// ---- _MSG/GVL_MSG_XTS.TcGVL
{attribute 'qualified_only'}
VAR_GLOBAL CONSTANT
  //-----------------------------------------------------------------------------
  // file paths for message system
  //  - compiler define option WIN switches to Windows file paths
  //-----------------------------------------------------------------------------
{IF defined (WIN)}
  {info 'WIN folders'}
  LOG_DIR               : STRING  := 'C:\TwinCAT\#MsgFiles\';       // delimiter at the end is mandatory!!
  CON_DIR               : STRING  := 'C:\TwinCAT\#Configuration\';  // delimiter at the end is mandatory!!
{ELSE}
  {info 'BSD folders'}
  LOG_DIR               : STRING  := '/usr/local/etc/TwinCAT/#MsgFiles/';       // delimiter at the end is mandatory!!
  CON_DIR               : STRING  := '/usr/local/etc/TwinCAT/#Configuration/';  // delimiter at the end is mandatory!!
{END_IF}

  LOG_FILE              : STRING  := 'MSG_XtsTransport_';
  LOG_FILE_APP          : STRING  := 'MSG_Application_';
  LOG_FILE_METRIC       : STRING  := 'MSG_XtsTransportMetrics_';

  MAX_MESSAGE           : UINT    := 2000; // max entry in message list
END_VAR
VAR_GLOBAL
  //-----------------------------------------------------------------------------
  // Message System
  //  - Everybody uses f_MessageSet(ST_Message)
  //    - DECISION WHICH LIST IS MADE IN f_MessageSet !!
  //    - which list to use is determined by e_Device in your message
  //
  //  - MessageData instances are self sufficient and need only 
  //    datafield assignment for correct data-flow
  //
  //
  //-----------------------------------------------------------------------------
  //-----------------------------------------------------------------------------
  //-----------------------------------------------------------------------------
  // (ST_Message.eDevice := e_Device.Application)
  //----------------------------------------------------------------------------- 
  ApplicationMessageData          : fb_MessageDataCtrl;
  ApplicationMessageCtrl          : st_message_ctrl;
  ApplicationMessageState         : st_message_state;

  ApplicationMessages             : ARRAY[1..MAX_MESSAGE] OF ST_Message;
  MessageApplicationIndex         : UINT := 0; // message index for higher layers (grouping, Instances, etc.)
  MessageApplicationError         : UINT := 0; // error counter for higher learning
  //-----------------------------------------------------------------------------
  //-----------------------------------------------------------------------------
  // (ST_Message.eDevice := from Device_Null to XfcAxis)
  //-----------------------------------------------------------------------------
  TransportMessageData            : fb_MessageDataCtrl;
  TransportMessageCtrl            : st_message_ctrl;
  TransportMessageState           : st_message_state;

  TransportMessages               : ARRAY[1..MAX_MESSAGE] OF ST_Message;
  MessageTransportIndex           : UINT := 0; // message index for base layer
  MessageTransportError           : UINT := 0; // error counter for base layer
  //-----------------------------------------------------------------------------
  //-----------------------------------------------------------------------------
  // (ST_Message.eDevice := e_Device.Metrics)
  //-----------------------------------------------------------------------------
  MetricsMessageData              : fb_MessageDataCtrl;
  MetricsMessageCtrl              : st_message_ctrl;
  MetricsMessageState             : st_message_state;

  MetricsMessages                 : ARRAY[1..MAX_MESSAGE] OF ST_Message;
  MessageMetricsIndex             : UINT := 0; // message index for metrics data
  MessageMetricsError             : UINT := 0; // error counter for metrics data
  //-----------------------------------------------------------------------------
  //-----------------------------------------------------------------------------
  // (ST_Message.eDevice := e_Device.ProductData)
  //-----------------------------------------------------------------------------
  ProductMessageData              : fb_MessageDataCtrl;   // This is for you
  ProductMessageCtrl              : st_message_ctrl;
  ProductMessageState             : st_message_state;

  ProductMessages                 : ARRAY[1..MAX_MESSAGE] OF ST_Message;
  MessageProductIndex             : UINT := 0; // message index for your product data
  MessageProductError             : UINT := 0; // error counter for your product data
  //-----------------------------------------------------------------------------
  //-----------------------------------------------------------------------------
  fbLocalTime                     : fb_LocalTime;
  dtLocalTime                     : DT;
  sLocalTime                      : STRING;
  //-----------------------------------------------------------------------------
  //-----------------------------------------------------------------------------
  //-----------------------------------------------------------------------------
  //-----------------------------------------------------------------------------
  MessageLevelXpu                 : E_MessageType;
  MessageLevelStations            : ARRAY[1..MAX_STATION] OF E_MessageType;
  MessageLevelMovers              : ARRAY[1..MAX_MOVER]   OF E_MessageType;

  MessageLevelProcess             : ARRAY[1..MAX_PROCESS] OF E_MessageType;

{IF defined (TEST)}
  {info 'TEST logging enabled'}
  MessageLevel                    : E_MessageType := eMessageinfo; // a lot of messages
{ELSE}
  MessageLevel                    : E_MessageType := eMessageEmpty; // only errors are written into list 
{END_IF}

END_VAR

// ---- _MSG/I_MessageData.TcIO
INTERFACE I_MessageData

PROPERTY DirRoot : POINTER to string(255)
SET
END_SET
END_PROPERTY

PROPERTY ErrorIndex : reference to uint
SET
END_SET
END_PROPERTY

PROPERTY FileRoot : pointer to string(255)
SET
END_SET
END_PROPERTY

PROPERTY LocalTime : pointer to DT
SET
END_SET
END_PROPERTY

PROPERTY MessageIndex : reference to uint
SET
END_SET
END_PROPERTY

PROPERTY MsgList : pointer to ARRAY[1..GVL_MSG_XTS.MAX_MESSAGE] OF st_message
SET
END_SET
END_PROPERTY

END_INTERFACE

// ---- _XML/Configuration/I_Configuration_Station.TcIO
INTERFACE I_Configuration_Station

METHOD Check : BOOL
END_METHOD

METHOD PRIVATE Cmd : E_DATA_STATE
VAR_INPUT
  Ctrl      : E_DATA_CTRL;
END_VAR
END_METHOD

PROPERTY Ctrl : REFERENCE to ST_DATA_CTRL
SET
END_SET
END_PROPERTY

PROPERTY Identity : OTCID
GET
END_GET
SET
END_SET
END_PROPERTY

PROPERTY State : REFERENCE TO ST_DATA_STATE
SET
END_SET
END_PROPERTY

PROPERTY StationParameter : pointer to ARRAY[1..MAX_STATION] OF ST_STATION_PARAMETER
SET
END_SET
END_PROPERTY

END_INTERFACE

// ---- APPLICATION/fb_Simulation.TcPOU
//---------------------------------------------------------------------------------------------------------------
//
//  HAUD 2023.03.27
//
//
//  fb_Simulation
//
//    !!! NOT FOR USE IN PRODUCTION !!! --> build something from your mind, this gets messy if you do not
//
//  - grouping of xts stations to sync start process
//  - nFirst to nLast xts stations are checked for starting process simultaneously
//  - basic preparation of station target index in PrepareTarget()
//  - handshake with station control for mover transport through station
//
//---------------------------------------------------------------------------------------------------------------
// This SOFTWARE is provided as an Exemple by THE PROVIDER "as is" and "with all faults." THE PROVIDER makes no 
// representations or warranties of any kind concerning the safety, suitability, lack of viruses, inaccuracies, 
// typographical errors, or other harmful components of this SOFTWARE. There are inherent dangers in the use of 
// any software, and you are solely responsible for determining whether this SOFTWARE is compatible with your 
// equipment and other software installed on your equipment. You are also solely responsible for the protection 
// of your equipment and backup of your data, and THE PROVIDER will not be liable for any damages you may suffer 
// in connection with using, modifying, or distributing this SOFTWARE.
//---------------------------------------------------------------------------------------------------------------
FUNCTION_BLOCK fb_Simulation
VAR
  _nProcessId                 : UINT;

  _sCheck                     : STRING;
  _tonProcess                 : Tc2_Standard.TON;
  _tProcess                   : TIME := T#500MS;

  _AllStationMoverPerMinute   : UDINT;
  _nMoverCountTotal           : UDINT;

  _tonPartsPerMinute          : Tc2_Standard.TON;

  {attribute 'displaymode':='bin'}
  _wEnter                     : DWORD;
  {attribute 'displaymode':='bin'}
  _wStart                     : DWORD;
  {attribute 'displaymode':='bin'}
  _wOut                       : DWORD;
  {attribute 'displaymode':='bin'}
  _wGone                      : DWORD;
  {attribute 'displaymode':='bin'}
  _wEnableProcess             : DWORD; // bits switch on stations

  {attribute 'displaymode':='bin'}
  _TargetMask                 : BYTE;

  _stCtrl                     : POINTER TO ARRAY[1..MAX_STATION]  OF ST_STATION_CTRL;
  _stState                    : POINTER TO ARRAY[1..MAX_STATION]  OF ST_STATION_STATE;

  // controlling bits from properties used on the outside
  _bNext,
  _bMoverEnter,
  _bMoverOut                  : BOOL;

  // who is included in process
  // _nFirst to _nLast MUST be in closed consecutive order
  _nProcessState,
  _nStation,
  _nStationCount,
  _nFirstStation,
  _nLastStation               : UINT;

  _nTarget,
  _nFirstTarget,
  _nLastTarget                : UINT;

  _nPreparedTarget            : ARRAY[1..MAX_MOVER]  OF UINT;

  _nMoverCountStartOld,
  _nMoverCountEnterOld,
  _nMoverCountEnter,
  _nMoverCountStart,
  _nMoverPerMinute,
  _nMoverCount,
  _nMoverCountOld             : ARRAY[1..MAX_STATION]  OF UDINT;

  _rCheckRangeLow,
  _rCheckRangeHigh            : LREAL; // position range the mover has to be in for infeed or sending to happen.

  _MessageLevel               : E_MessageType;
  _stMsg                      : ST_Message;
END_VAR

METHOD Check : BOOL

IF (_nFirstStation < 1) OR
   (_nFirstStation > MAX_STATION)
THEN
  _sCheck                     := '_nFirstStation out of bounds';
  RETURN;
END_IF

IF (_nLastStation < 1) OR
   (_nLastStation > MAX_STATION)
THEN
  _sCheck                     := '_nLastStation out of bounds';
  RETURN;
END_IF

IF (_nFirstTarget < 1) OR
   (_nFirstTarget > MAX_STATION)
THEN
  _sCheck                     := '_nFirstTarget out of bounds';
  RETURN;
END_IF

IF (_nLastTarget < 1) OR
   (_nLastTarget > MAX_STATION)
THEN
  _sCheck                     := '_nLastTarget out of bounds';
  RETURN;
END_IF

IF NOT (_stCtrl  <> 0)
THEN
  _sCheck                     := '_stCtrl: missing pointer';
  RETURN;
END_IF

IF NOT (_stState <> 0)
THEN
  _sCheck                     := '_stState: missing pointer';
  RETURN;
END_IF


_sCheck                       := TO_STRING(E_PROGRESS.PROGRESS_DONE);
Check                         := TRUE;
END_METHOD

PROPERTY CheckRangeHigh : lreal
GET
CheckRangeHigh := _rCheckRangeHigh;
END_GET
SET
_rCheckRangeHigh := CheckRangeHigh;
END_SET
END_PROPERTY

PROPERTY CheckRangeLow : lreal
GET
CheckRangeLow := _rCheckRangeLow;
END_GET
SET
_rCheckRangeLow := CheckRangeLow;
END_SET
END_PROPERTY

METHOD Cycle
VAR_INST
  _interAllStationsCounter    : UDINT;

  _rtrigProcessEnter,
  _rtrigProcessStart,
  _rtrigProcess       : ARRAY[1..MAX_STATION] OF Tc2_Standard.R_TRIG;

  _k                  : UINT;
  _wEnable            : DWORD;
END_VAR
//-----------------------------------------------------------------------------------------------------------------
IF NOT Check() THEN RETURN; END_IF
//-----------------------------------------------------------------------------------------------------------------
_nStationCount                              := _nLastStation - _nFirstStation + 1;
//-----------------------------------------------------------------------------------------------------------------
//-----------------------------------------------------------------------------------------------------------------
IF (_nStationCount < 1)
THEN
  RETURN;
END_IF
//-----------------------------------------------------------------------------------------------------------------
//-----------------------------------------------------------------------------------------------------------------
FOR _nStation := _nLastStation TO _nFirstStation BY(-1) 
DO
  CASE _stState^[_nStation].State
  OF
    //-------------------------------------------------------------------------------------------------------------
    E_STATION_STATE.STATION_DISABLE,
    E_STATION_STATE.STATION_ENABLE, 
    E_STATION_STATE.STATION_DETECT_MOVER:
      _wStart   := _wOut    := _wGone       := 0;
      _wEnter                               := DelBit(_wEnter, (_nStation-_nFirstStation));
      IF (GetBit(_wEnableProcess, (_nStation-_nFirstStation)))
      THEN
        IF (_bMoverEnter)
        THEN
          _stCtrl^[_nStation].Cmd           := E_STATION_CTRL.STATION_ENABLE;
        ELSE
          _stCtrl^[_nStation].Cmd           := E_STATION_CTRL.STATION_DISABLE;
        END_IF
      ELSE
        _stCtrl^[_nStation].Cmd             := E_STATION_CTRL.STATION_DISABLE;
      END_IF


    //-------------------------------------------------------------------------------------------------------------
    E_STATION_STATE.STATION_MOVER_ENTER:
      _wEnter                               := SetBit(_wEnter, (_nStation-_nFirstStation));
      IF _bMoverEnter
      THEN
        _tonProcess(IN                      := FALSE, 
                    PT                      := _tProcess);

        _stCtrl^[_nStation].nTargetStation  := 0;

        IF (_tProcess < T#10MS)
        THEN
          IF (_rCheckRangeHigh > _rCheckRangeLow)
          THEN
            IF (_stState^[_nStation].rMoverModPos > _rCheckRangeLow) AND
               (_stState^[_nStation].rMoverModPos < _rCheckRangeHigh)
            THEN
              _stCtrl^[_nStation].Cmd       := E_STATION_CTRL.STATION_MOVER_SEND;
            END_IF
          ELSE
            IF (_stState^[_nStation].rMoverModPos > _rCheckRangeLow) OR
               (_stState^[_nStation].rMoverModPos < _rCheckRangeHigh)
            THEN
              _stCtrl^[_nStation].Cmd       := E_STATION_CTRL.STATION_MOVER_SEND;
            END_IF
          END_IF
        ELSE
          IF (_rCheckRangeHigh > _rCheckRangeLow)
          THEN
            IF (_stState^[_nStation].rMoverModPos > _rCheckRangeLow) AND
               (_stState^[_nStation].rMoverModPos < _rCheckRangeHigh)
            THEN
              _stCtrl^[_nStation].Cmd       := E_STATION_CTRL.STATION_MOVER_ENTER;
            END_IF
          ELSE
            IF (_stState^[_nStation].rMoverModPos > _rCheckRangeLow) OR
               (_stState^[_nStation].rMoverModPos < _rCheckRangeHigh)
            THEN
              _stCtrl^[_nStation].Cmd       := E_STATION_CTRL.STATION_MOVER_ENTER;
            END_IF
          END_IF
        END_IF
      END_IF

    //-------------------------------------------------------------------------------------------------------------
    E_STATION_STATE.STATION_PROCESS_START:
      _wEnter                               := DelBit(_wEnter, (_nStation-_nFirstStation));
      _wStart                               := SetBit(_wStart, (_nStation-_nFirstStation));
  
      // check if ALL XtsStations have mover in place to work
      IF (_wStart = _wEnableProcess)
      THEN
        _tonProcess(IN                      := TRUE, 
                    PT                      := _tProcess);

        IF _tonProcess.Q
        THEN
          PrepareTargets(FALSE);
          _stCtrl^[_nStation].Cmd           := E_STATION_CTRL.STATION_PROCESS_DONE;
        END_IF
      END_IF

    //-------------------------------------------------------------------------------------------------------------
    E_STATION_STATE.STATION_CHECK_NEST:
      _wEnter                               := SetBit(_wEnter, (_nStation-_nFirstStation));
      _wStart                               := DelBit(_wStart, (_nStation-_nFirstStation));
      _tonProcess(IN                        := FALSE, 
                  PT                        := _tProcess);

      IF (_bNext)
      THEN
        // check if ALL XtsStations have nest to work
        IF (_wEnter = _wEnableProcess)
        THEN
          _stCtrl^[_nStation].Cmd           := E_STATION_CTRL.STATION_MOVER_ENTER;
        END_IF
      END_IF

    //-------------------------------------------------------------------------------------------------------------
    E_STATION_STATE.STATION_MOVER_OUT:
      _wOut                                 := SetBit(_wOut, (_nStation-_nFirstStation));
      _tonProcess(IN                        := FALSE, 
                  PT                        := _tProcess);

      IF _bMoverOut
      THEN
        // nest mask for this mover in target station, sender decides what to work in target
        _stCtrl^[_nStation].nMask           := _TargetMask;

        // check if ALL XtsStations have mover to send
        IF (_wOut = _wEnableProcess)
        THEN
          _nProcessState                    := 10;
        END_IF
      END_IF
  END_CASE
END_FOR
//-----------------------------------------------------------------------------------------------------------------
//-----------------------------------------------------------------------------------------------------------------
CASE _nProcessState
OF
10:
  // ctrl has to decide where to send mover; this depends on YOUR decision
  IF PrepareTargets(TRUE)
  THEN
    PrepareTargets(FALSE);
    _nProcessState                          := 30;
  END_IF
END_CASE
CASE _nProcessState
OF
30:
  FOR _nStation := _nLastStation TO _nFirstStation BY(-1) 
  DO
    IF _bNext
    THEN
      // start outfeed of mover
      _stCtrl^[_nStation].Cmd               := E_STATION_CTRL.STATION_MOVER_OUT;
    END_IF

    CASE _stState^[_nStation].State
    OF
      E_STATION_STATE.STATION_MOVER_GONE:
        _wStart   := _wEnter                := 0;
        // whO is gone?
        _wGone                              := SetBit(_wGone, (_nStation-_nFirstStation));
    END_CASE
  END_FOR
  // check if ALL XtsStations are empty
  IF (_wGone = _wEnableProcess)
  THEN
    _nProcessState                          := 40;
    IF (_MessageLevel > E_MessageType.eMessageVerbose)
    THEN
      _stMsg.eType                          := E_MessageType.eMessageSentient;
      _stMsg.eDevice                        := e_Device.Metrics + TO_UINT(_nProcessId);
      _stMsg.eSubdevice                     := e_Subdevice.Process_StationCollector;
      _stMsg.iErrorNumber                   := _nProcessId;
      _stMsg.sText                          := concat('ALL MOVER: ', TO_STRING(E_STATION_STATE.STATION_MOVER_GONE));

      f_MessageSet(_stMsg);
    END_IF
  END_IF
END_CASE
CASE _nProcessState
OF
40:
  _nProcessState                            := 0;
  FOR _nStation := _nLastStation TO _nFirstStation BY(-1) 
  DO
    // let XtsStations jump back to disable
    _stCtrl^[_nStation].Cmd                 := E_STATION_CTRL.STATION_MOVER_GONE;
  END_FOR
END_CASE
//-----------------------------------------------------------------------------------------------------------------
//-----------------------------------------------------------------------------------------------------------------
//-----------------------------------------------------------------------------------------------------------------
// Mover per Minute counter all XtsStations in range
//-----------------------------------------------------------------------------------------------------------------
_nMoverCountTotal                           :=
_AllStationMoverPerMinute                   := 0; 
//-----------------------------------------------------------------------------------------------------------------
// mover counter
//-----------------------------------------------------------------------------------------------------------------
FOR _k := _nLastStation TO _nFirstStation BY(-1)
DO
  //---------------------------------------------------------------------------------------------------------------
  _rtrigProcess[_k](CLK:= ( _stCtrl^[_k].Cmd = E_STATION_CTRL.STATION_MOVER_OUT));
  //---------------------------------------------------------------------------------------------------------------
  IF _rtrigProcess[_k].Q
  THEN
    _nMoverCount[_k]                        := _nMoverCount[_k] + 1;

    IF (_MessageLevel > E_MessageType.eMessageError)
    THEN
      _stMsg.eType                          := E_MessageType.eMessageInfo;
      _stMsg.eDevice                        := e_Device.Metrics + TO_UINT(_nProcessId);
      _stMsg.eSubdevice                     := e_Subdevice.Process_StationCollector;
      _stMsg.iErrorNumber                   := _k;
      _stMsg.sText                          := concat('MoverCountStation[ ]: ', TO_STRING(_nMoverCount[_k]));
      _stMsg.sText                          := concat(_stMsg.sText, ': E_STATION_CTRL.');
      _stMsg.sText                          := concat(_stMsg.sText, TO_STRING(_stCtrl^[_k].Cmd));
      f_MessageSet(_stMsg);
    END_IF
  END_IF

  //---------------------------------------------------------------------------------------------------------------
  _rtrigProcessStart[_k](CLK:= ( _stState^[_k].State = E_STATION_STATE.STATION_PROCESS_START));
  //---------------------------------------------------------------------------------------------------------------
  IF _rtrigProcessStart[_k].Q
  THEN
    _nMoverCountStart[_k]                   := _nMoverCountStart[_k] + 1;

    IF (_MessageLevel > E_MessageType.eMessageInfo)
    THEN
      _stMsg.eType                          := E_MessageType.eMessageVerbose;
      _stMsg.eDevice                        := e_Device.Metrics + TO_UINT(_nProcessId);
                            
      _stMsg.eSubdevice                     := e_Subdevice.Process_StationCollector;
      _stMsg.iErrorNumber                   := _k;
      _stMsg.sText                          := concat('MoverCountStation[ ]: ', TO_STRING(_nMoverCountEnter[_k]));
      _stMsg.sText                          := concat(_stMsg.sText, ': E_STATION_STATE.');
      _stMsg.sText                          := concat(_stMsg.sText, TO_STRING(_stState^[_k].State));
      f_MessageSet(_stMsg);
    END_IF
  END_IF

  //---------------------------------------------------------------------------------------------------------------
  _rtrigProcessEnter[_k](CLK:= ( _stCtrl^[_k].Cmd = E_STATION_CTRL.STATION_MOVER_ENTER));
  //---------------------------------------------------------------------------------------------------------------
  IF _rtrigProcessEnter[_k].Q
  THEN
    _nMoverCountEnter[_k]                   := _nMoverCountEnter[_k] + 1;

    IF (_MessageLevel > E_MessageType.eMessageVerbose)
    THEN
      _stMsg.eType                          := E_MessageType.eMessageSentient;
      _stMsg.eDevice                        := e_Device.Metrics + TO_UINT(_nProcessId);
                            
      _stMsg.eSubdevice                     := e_Subdevice.Process_StationCollector;
      _stMsg.iErrorNumber                   := _k;
      _stMsg.sText                          := concat('MoverCountStation[ ]: ', TO_STRING(_nMoverCountEnter[_k]));
      _stMsg.sText                          := concat(_stMsg.sText, ': E_STATION_CTRL.');
      _stMsg.sText                          := concat(_stMsg.sText, TO_STRING(_stCtrl^[_k].Cmd));
      f_MessageSet(_stMsg);
    END_IF
  END_IF
  //---------------------------------------------------------------------------------------------------------------
  //---------------------------------------------------------------------------------------------------------------
  IF _tonPartsperMinute.Q
  THEN
    // count every XtsStation in range
    _nMoverPerMinute[_k]                    := _nMoverCount[_k] - _nMoverCountOld[_k];
    _nMoverCountOld [_k]                    := _nMoverCount[_k];

    _nMoverCountEnterOld [_k]               := _nMoverCountEnter[_k];
    _nMoverCountStartOld [_k]               := _nMoverCountStart[_k];
  END_IF
  // sum up all XtsStations in range
  _AllStationMoverPerMinute                 := _AllStationMoverPerMinute + _nMoverPerMinute[_k]; 
  _interAllStationsCounter                  := _AllStationMoverPerMinute + _nMoverPerMinute[_k];

  // sum up all mover counts in range
  _nMoverCountTotal                         := _nMoverCountTotal + _nMoverCount[_k];
END_FOR
//-----------------------------------------------------------------------------------------------------------------
//-----------------------------------------------------------------------------------------------------------------
// total mover per minute message for all stations in this process
//-----------------------------------------------------------------------------------------------------------------
//-----------------------------------------------------------------------------------------------------------------
IF _tonPartsperMinute.q
THEN
  _tonPartsperMinute(IN:=FALSE);

  IF (_MessageLevel > E_MessageType.eMessageError)
  THEN
    _stMsg.eType                          := E_MessageType.eMessageBatch;
    _stMsg.eDevice                        := e_Device.Metrics + TO_UINT(_nProcessId);
  
    _stMsg.eSubdevice                     := e_Subdevice.Process_StationCollector;
    _stMsg.iErrorNumber                   := _nMoverCountTotal;
    _stMsg.sText                          := concat('MoverCountTotal: ', TO_STRING(_nMoverCountTotal));
    _stMsg.sText                          := concat(_stMsg.sText, ': StationLast: ');
    _stMsg.sText                          := concat(_stMsg.sText, TO_STRING(_nLastStation));
    _stMsg.sText                          := concat(_stMsg.sText, ': StationFirst: ');
    _stMsg.sText                          := concat(_stMsg.sText, TO_STRING(_nFirstStation));
    f_MessageSet(_stMsg);
  END_IF
END_IF
//-----------------------------------------------------------------------------------------------------------------
_tonPartsperMinute(IN:= TRUE,   PT:= T#60S);
//-----------------------------------------------------------------------------------------------------------------
//-----------------------------------------------------------------------------------------------------------------
END_METHOD

METHOD PUBLIC DelBit : DWORD
VAR_INPUT
  inVal   : DWORD;
  bitNo   : DINT;
END_VAR
VAR
  wConst : dWORD := 1;
END_VAR
IF ( inVal AND SHL( wConst,bitNo MOD 32 ) ) > 0 THEN
  DelBit := inVal XOR (SHL( wConst,bitNo MOD 32 ));
ELSE
  DelBit := inVal;
END_IF
END_METHOD

METHOD Disable : BOOL
VAR_INPUT
END_VAR
IF NOT (_nLastStation   > 0) OR
   NOT (_nFirstStation  > 0) OR
   NOT (_nLastStation   < MAX_STATION+1) OR
   NOT (_nFirstStation  < MAX_STATION+1)
THEN
  Disable := FALSE;
ELSE
  FOR _nStation := _nLastStation TO _nFirstStation BY(-1) 
  DO
    _stCtrl^[_nStation].Cmd               := E_STATION_CTRL.STATION_DISABLE;
    _stCtrl^[_nStation].nMask             := 0;
  END_FOR

  memset(ADR(_nMoverCount),    0, SIZEOF(_nMoverCount));
  memset(ADR(_nMoverCountOld), 0, SIZEOF(_nMoverCountOld));
  _nProcessState :=  _nTarget             := 0;
  
  Disable := TRUE;
END_IF
END_METHOD

PROPERTY EnableProcess : dword
GET
EnableProcess := _wEnableProcess;
END_GET
SET
_wEnableProcess := EnableProcess;
END_SET
END_PROPERTY

METHOD PUBLIC GetBit : BOOL
VAR_INPUT
  inVal   : DWORD;
  bitNo   : DINT;
END_VAR
VAR
  wConst : DWORD := 1;
END_VAR
IF ( inVal AND SHL( wConst,DINT_TO_SINT(bitNo) MOD 32 ) ) > 0
THEN
  GetBit := TRUE;
ELSE
  GetBit := FALSE;
END_IF
END_METHOD

METHOD Init : BOOL
VAR_INPUT
END_VAR
IF NOT (_nLastStation   > 0) OR
   NOT (_nFirstStation  > 0) OR
   NOT (_nLastStation   < MAX_STATION+1) OR
   NOT (_nFirstStation  < MAX_STATION+1)
THEN
  Init := FALSE;
ELSE
  FOR _nStation := _nLastStation TO _nFirstStation BY(-1) 
  DO
    _stCtrl^[_nStation].Cmd               := E_STATION_CTRL.STATION_INIT;
    _stCtrl^[_nStation].nMask             := 0;
  END_FOR

  memset(ADR(_nMoverCount),    0, SIZEOF(_nMoverCount));
  memset(ADR(_nMoverCountOld), 0, SIZEOF(_nMoverCountOld));
  _nProcessState :=  _nTarget             := 0;
  
  Init := TRUE;
END_IF
END_METHOD

PROPERTY MessageLevel : e_MessageType
GET
MessageLevel := _MessageLevel;
END_GET
SET
VAR
  _ix : uint;
END_VAR
_MessageLevel := MessageLevel;
END_SET
END_PROPERTY

PROPERTY MoverEnter : bool
GET
MoverEnter := _bMoverEnter;
END_GET
SET
_bMoverEnter := MoverEnter;
END_SET
END_PROPERTY

PROPERTY MoverOut : bool
GET
MoverOut := _bMoverOut;
END_GET
SET
_bMoverOut := MoverOut;
END_SET
END_PROPERTY

METHOD Next : BOOL
VAR_INPUT
  Nxt  : Bool;
END_VAR
_bNext := Nxt;
END_METHOD

METHOD PRIVATE PrepareTargets : BOOL
VAR_INPUT
  Execute         : BOOL;
END_VAR
VAR_INST
  _idxStations    : uint;
  _nt,
  _nstate         : UINT;
END_VAR

IF NOT Check() THEN RETURN; END_IF

IF NOT Execute
THEN
  _nstate                             := 0;
END_IF


CASE _nstate
OF
  0:
    IF Execute
    THEN
      _nstate                         := 10;
    END_IF
END_CASE
CASE _nstate
OF
  10:
    _nstate                           := 20;

    FOR _idxStations := _nLastStation TO _nFirstStation BY(-1) 
    DO
      _nt                               := TO_USINT(_nLastTarget - _nTarget);
      _nTarget                          := _nTarget + 1;
  
      _nPreparedTarget[_stState^[_idxStations].nMoverId]  := _nt;
      _stCtrl^[_idxStations].nTargetStation               := TO_USINT(_nt);
  
      IF (_nLastTarget - _nTarget < _nFirstTarget)
      THEN
        _nTarget                        := 0;
      END_IF
    END_FOR
END_CASE
CASE _nstate
OF
  20:
    PrepareTargets                    := TRUE;
END_CASE
END_METHOD

PROPERTY ProcessId : uint
GET
ProcessId := _nProcessId;
END_GET
SET
_nProcessId := ProcessId;
END_SET
END_PROPERTY

PROPERTY ProcessTime : time
GET
ProcessTime := _tProcess;
END_GET
SET
_tProcess := ProcessTime;
END_SET
END_PROPERTY

METHOD PUBLIC SetBit : DWORD
VAR_INPUT
  inVal   : DWORD;
  bitNo   : DINT;
END_VAR
VAR
  wConst  : dWORD := 1;
END_VAR
SetBit := inVal OR SHL( wConst,bitNo MOD 32 );
END_METHOD

PROPERTY StationCount : uint
GET
StationCount := _nStationCount;
END_GET
END_PROPERTY

PROPERTY StationCtrl : pointer to ARRAY[1..MAX_STATION]  OF ST_STATION_CTRL;
SET
_stCtrl := StationCtrl;
END_SET
END_PROPERTY

PROPERTY StationFirst : uint
GET
StationFirst := _nFirstStation;
END_GET
SET
_nFirstStation := StationFirst;
END_SET
END_PROPERTY

PROPERTY StationLast : uint
GET
StationLast := _nLastStation;
END_GET
SET
_nLastStation := StationLast;
END_SET
END_PROPERTY

PROPERTY StationState : POINTER TO ARRAY[1..MAX_STATION]  OF ST_STATION_STATE
SET
_stState := StationState;
END_SET
END_PROPERTY

PROPERTY TargetFirst : uint
GET
TargetFirst := _nFirstTarget;
END_GET
SET
_nFirstTarget := TargetFirst;
END_SET
END_PROPERTY

PROPERTY TargetLast : uint
GET
TargetLast := _nLastTarget;
END_GET
SET
_nLastTarget := TargetLast;
END_SET
END_PROPERTY

PROPERTY TargetMask : byte
GET
TargetMask := _TargetMask;
END_GET
SET
_TargetMask := TargetMask;
END_SET
END_PROPERTY

END_FUNCTION_BLOCK

// ---- _MSG/f_MessageSet.TcPOU
FUNCTION f_MessageSet : BOOL
VAR_INPUT
  stMessage     : ST_Message;
END_VAR
VAR
  _uiIndex      : UINT;
  _MainDevice   : e_Device;
  _nModRes      : UDINT;     // residual after modulo
END_VAR

stMessage.tTime                     := GVL_MSG_XTS.sLocalTime;

// why here? so all calls to this function may stay the same
_nModRes                            := stMessage.eDevice MOD e_Device.General;
_MainDevice                         := stMessage.eDevice - _nModRes;

CASE _MainDevice
OF
  //--------------------------------------------------------------------------------
  e_device.DataProduct:
    // this is your data, if you choose to use this message system
    FOR _uiIndex := 1 TO GVL_MSG_XTS.MAX_MESSAGE
    DO
      IF (GVL_MSG_XTS.ProductMessages[_uiIndex].eType = e_MessageType.eMessageEmpty)
      THEN
        GVL_MSG_XTS.ProductMessages[_uiIndex]      := stMessage;
        GVL_MSG_XTS.MessageProductIndex            := _uiIndex;
        EXIT;
      END_IF
    END_FOR
  
    IF (stMessage.eType = E_MessageType.eMessageError)
    THEN
      // in case of error: increment counter
      GVL_MSG_XTS.MessageProductError              := GVL_MSG_XTS.MessageProductError + 1;
    END_IF
  //--------------------------------------------------------------------------------
  e_Device.Process,
  e_Device.Application:
    FOR _uiIndex := 1 TO GVL_MSG_XTS.MAX_MESSAGE
    DO
      IF (GVL_MSG_XTS.ApplicationMessages[_uiIndex].eType = e_MessageType.eMessageEmpty)
      THEN
        GVL_MSG_XTS.ApplicationMessages[_uiIndex]  := stMessage;    // yes, we grab global values directly, only here
        GVL_MSG_XTS.MessageApplicationIndex        := _uiIndex;
        EXIT;
      END_IF
    END_FOR
    IF (stMessage.eType = E_MessageType.eMessageError)
    THEN
      // in case of error: increment counter
      GVL_MSG_XTS.MessageApplicationError          := GVL_MSG_XTS.MessageApplicationError + 1;
    END_IF
  //--------------------------------------------------------------------------------
  e_Device.MetricsXts:
    FOR _uiIndex := 1 TO GVL_MSG_XTS.MAX_MESSAGE
    DO
      IF (GVL_MSG_XTS.MetricsMessages[_uiIndex].eType = e_MessageType.eMessageEmpty)
      THEN
        GVL_MSG_XTS.MetricsMessages[_uiIndex]      := stMessage;    // yes, we grab global values directly, only here
        GVL_MSG_XTS.MessageMetricsIndex            := _uiIndex;
        EXIT;
      END_IF
    END_FOR
    IF (stMessage.eType = E_MessageType.eMessageError)
    THEN
      // in case of error: increment counter
      GVL_MSG_XTS.MessageMetricsError              := GVL_MSG_XTS.MessageMetricsError + 1;
    END_IF
  //--------------------------------------------------------------------------------
  e_Device.MetricsAxis:
    FOR _uiIndex := 1 TO GVL_MSG_XTS.MAX_MESSAGE
    DO
      IF (GVL_MSG_AXIS.MetricMessages[_uiIndex].eType = e_MessageType.eMessageEmpty)
      THEN
        GVL_MSG_AXIS.MetricMessages[_uiIndex]  := stMessage;    // yes, we grab global values directly, only here
        GVL_MSG_AXIS.MessageMetricIndex        := _uiIndex;
        EXIT;
      END_IF
    END_FOR
    IF (stMessage.eType = E_MessageType.eMessageError)
    THEN
      // in case of error: increment counter
      GVL_MSG_AXIS.MessageMetricError          := GVL_MSG_AXIS.MessageMetricError + 1;
    END_IF
  //--------------------------------------------------------------------------------
  e_Device.Axis,
  e_Device.XfcAxis,
  e_device.XfcTouchProbe,
  e_device.XfcTriggerBox,
  e_Device.Camming,
  e_device.NciChannel,
  e_device.NciChannelCtrl:
    FOR _uiIndex := 1 TO GVL_MSG_XTS.MAX_MESSAGE
    DO
      IF (GVL_MSG_AXIS.MotionMessages[_uiIndex].eType = e_MessageType.eMessageEmpty)
      THEN
        GVL_MSG_AXIS.MotionMessages[_uiIndex]  := stMessage;    // yes, we grab global values directly, only here
        GVL_MSG_AXIS.MessageMotionIndex        := _uiIndex;
        EXIT;
      END_IF
    END_FOR
    IF (stMessage.eType = E_MessageType.eMessageError)
    THEN
      // in case of error: increment counter
      GVL_MSG_AXIS.MessageMotionError           := GVL_MSG_AXIS.MessageMotionError + 1;
    END_IF
  //--------------------------------------------------------------------------------
ELSE
  CASE stMessage.eDevice
  OF
    Device_MainApplication,
    Device_XmlData,              
    Device_Utilities:
      FOR _uiIndex := 1 TO GVL_MSG_XTS.MAX_MESSAGE
      DO
        IF (GVL_MSG_XTS.ApplicationMessages[_uiIndex].eType = e_MessageType.eMessageEmpty)
        THEN
          GVL_MSG_XTS.ApplicationMessages[_uiIndex]:= stMessage;    // yes, we grab global values directly, only here
          GVL_MSG_XTS.MessageApplicationIndex      := _uiIndex;
          EXIT;
        END_IF
      END_FOR
      IF (stMessage.eType = E_MessageType.eMessageError)
      THEN
        // in case of error: increment counter
        GVL_MSG_XTS.MessageApplicationError        := GVL_MSG_XTS.MessageApplicationError + 1;
      END_IF

    Device_MainAxis,
    Device_Nci,
    Device_Cam,
    Device_Functions,
    Device_FlyingSaw,
    Device_ParameterSelector:     // PLC_MOTION
      FOR _uiIndex := 1 TO GVL_MSG_XTS.MAX_MESSAGE
      DO
        IF (GVL_MSG_AXIS.MotionMessages[_uiIndex].eType = e_MessageType.eMessageEmpty)
        THEN
          GVL_MSG_AXIS.MotionMessages[_uiIndex]:= stMessage;    // yes, we grab global values directly, only here
          GVL_MSG_AXIS.MessageMotionIndex      := _uiIndex;
          EXIT;
        END_IF
      END_FOR
      IF (stMessage.eType = E_MessageType.eMessageError)
      THEN
        // in case of error: increment counter
        GVL_MSG_AXIS.MessageMotionError        := GVL_MSG_AXIS.MessageMotionError + 1;
      END_IF

    Device_Main,
    Device_MoverSelector:
      FOR _uiIndex := 1 TO GVL_MSG_XTS.MAX_MESSAGE
      DO
        IF (GVL_MSG_XTS.TransportMessages[_uiIndex].eType = e_MessageType.eMessageEmpty)
        THEN
          GVL_MSG_XTS.TransportMessages[_uiIndex]  := stMessage;
          GVL_MSG_XTS.MessageTransportIndex        := _uiIndex;
          EXIT;
        END_IF
      END_FOR
  ELSE    
    //--------------------------------------------------------------------------------
    FOR _uiIndex := 1 TO GVL_MSG_XTS.MAX_MESSAGE
    DO
      IF (GVL_MSG_XTS.TransportMessages[_uiIndex].eType = e_MessageType.eMessageEmpty)
      THEN
        GVL_MSG_XTS.TransportMessages[_uiIndex]    := stMessage;
        GVL_MSG_XTS.MessageTransportIndex          := _uiIndex;
        EXIT;
      END_IF
    END_FOR
  
    IF (stMessage.eType = E_MessageType.eMessageError)
    THEN
      // in case of error: increment counter
      GVL_MSG_XTS.MessageTransportError := GVL_MSG_XTS.MessageTransportError + 1;
    END_IF
  END_CASE
END_CASE

END_FUNCTION

// ---- _MSG/class/fb_MessageDataCtrl.TcPOU
FUNCTION_BLOCK fb_MessageDataCtrl EXTENDS fb_MessageData
VAR
  _stCtrl       : REFERENCE TO ST_MESSAGE_CTRL;
  _stState      : REFERENCE TO ST_MESSAGE_STATE;

  _eCmd,
  _eCmdOld      : E_MESSAGE_CTRL;

  _eResult,
  _eJobResult   : E_PROGRESS;

  _eState       : E_MESSAGE_STATE;

END_VAR

//-----------------------------------------------------------------------------
// check pointers
//-----------------------------------------------------------------------------
IF NOT Check()
THEN
  _eResult                      := E_PROGRESS.PROGRESS_ERROR;
  RETURN;
END_IF
//-----------------------------------------------------------------------------
// check date
// new message file for a new day
//-----------------------------------------------------------------------------
IF (FolderDate(_dtLocalTime) <> _sFolderDate)
THEN
  _bFileCreated                 := FALSE;
END_IF
//-----------------------------------------------------------------------------
//----------------------------------------------------------------------------- 
// copy to local for debug
_eCmd                         := _stCtrl.Cmd;

// cyclic check for command change
// get state for cmd
IF (_eCmd <> _eCmdOld)
THEN
  // get matching sdtate for Ctrl.Cmd
  _eState                     := Cmd(_eCmd);
  _eCmdOld                    := _eCmd;
END_IF


CASE _eResult
OF
  E_PROGRESS.PROGRESS_INVALID:
    _stState.State            := E_MESSAGE_STATE.MSG_STATE_NULL;

  E_PROGRESS.PROGRESS_ERROR:
    _stState.State            := _eState + E_PROGRESS.PROGRESS_ERROR;

  E_PROGRESS.PROGRESS_DONE:
    _stState.State            := _eState + E_PROGRESS.PROGRESS_DONE;

ELSE
  // work in progress
  // update progress for extern use
  _stState.State              := _eState + _eResult;

  CASE _eState
  OF
    E_MESSAGE_STATE.MSG_STATE_INIT:
      _eResult                := BuildFolder(TRUE);


    E_MESSAGE_STATE.MSG_STATE_IDLE:
      IF (_nMsgIndex < GVL_MSG_XTS.MAX_MESSAGE - GVL_MSG_XTS.MAX_MESSAGE/10)
      THEN
        _eResult              := E_PROGRESS.PROGRESS_WORKING;
      ELSE
        _eResult              := E_PROGRESS.PROGRESS_DONE;
        _nMsgIndex            := 0;
        // copy from attached list to local
        memcpy(ADR(_aWriteList), _pMsgList, SIZEOF(_aWriteList));
        // clear attached list
        memset(_pMsgList, 0, SIZEOF(_aWriteList));
      END_IF


    E_MESSAGE_STATE.MSG_STATE_WRITE:
      _eResult                := BuildFileData(TRUE);

  ELSE
      _eResult               := E_PROGRESS.PROGRESS_INVALID;
  END_CASE
END_CASE

METHOD BuildFileData : e_progress
VAR_INPUT
  Execute     : BOOL;
END_VAR
VAR_INST
  _nErrorId   : UDINT;
  _eState,
  _eRes       : E_PROGRESS;
  _eFlow      : E_MESSAGE_FLOW;

  _nStringLength  : UINT;
END_VAR
//-----------------------------------------------------------------------------
IF NOT Execute 
THEN
  _eRes                           := WriteData(FALSE);
  _eRes                           := BuildFolder(FALSE);
	_eState                         := E_PROGRESS.PROGRESS_INIT; 
END_IF 
//-----------------------------------------------------------------------------
IF NOT Check() 
THEN 
	BuildFileData                   := E_PROGRESS.PROGRESS_ERROR; 
	RETURN; 
END_IF
//-----------------------------------------------------------------------------
//-----------------------------------------------------------------------------
CASE _eState
OF
  E_PROGRESS.PROGRESS_INIT:
    IF Execute
    THEN
      _nErrorId                   := 0;
      _iStart 	                  := 1;
      _iEnd 		                  := SEL((_nMsgIndex > GVL_MSG_XTS.MAX_MESSAGE-1),
                                          _nMsgIndex,
                                          GVL_MSG_XTS.MAX_MESSAGE);

      memset(ADR(_sWriteData),0,SIZEOF(_sWriteData));

      IF (_sFolderDate <> FolderDate(_dtLocalTime))
      THEN
        _eState                   := E_PROGRESS.PROGRESS_PREPARE;
      ELSE
        _eState                   := E_PROGRESS.PROGRESS_BUSY;
        _eFlow                    := E_MESSAGE_FLOW.MSG_FLOW_LINE_START;
      END_IF
    END_IF
END_CASE
//-----------------------------------------------------------------------------
//-----------------------------------------------------------------------------
CASE _eState
OF
  E_PROGRESS.PROGRESS_PREPARE:
    _eRes                         := BuildFolder(TRUE);
    CASE _eRes
    OF
      E_PROGRESS.PROGRESS_DONE:
      _eState                     := E_PROGRESS.PROGRESS_BUSY;
      _eFlow                      := E_MESSAGE_FLOW.MSG_FLOW_LINE_START;

      E_PROGRESS.PROGRESS_ERROR:
      _eState                     := E_PROGRESS.PROGRESS_ERROR;
    END_CASE
END_CASE
//-----------------------------------------------------------------------------
//-----------------------------------------------------------------------------
CASE _eState
OF
  E_PROGRESS.PROGRESS_BUSY:
  CASE _eFlow
  OF
    E_MESSAGE_FLOW.MSG_FLOW_LINE_START:
      _eRes                       := BuildFolder(FALSE);
      _nErrIndex                  := 0; // rise and shine, all quarrels erased but not forgotten
      _nMsgIndex                  := 0;
  
      // copy from attached list to local
      memcpy(ADR(_aWriteList), _pMsgList, SIZEOF(_aWriteList));
  
      // clear attached list
      memset(_pMsgList, 0, SIZEOF(_aWriteList));


      _eFlow                      := E_MESSAGE_FLOW.MSG_FLOW_LINE_BUILD;
      _iCount                     := _iStart;
  END_CASE
  CASE _eFlow
  OF
    E_MESSAGE_FLOW.MSG_FLOW_LINE_BUILD:
      _eFlow                      := E_MESSAGE_FLOW.MSG_FLOW_LINE_CHECK;
      IF (_aWriteList[_iCount].eType > E_MessageType.eMessageEmpty)
      THEN
        _sTmp                     := TO_STRING(_aWriteList[_iCount].eType);
        _sTmp                     := Tc2_Standard.CONCAT(_sTmp, _sTab);
        _sTmp                     := Tc2_Standard.CONCAT(_sTmp, _aWriteList[_iCount].tTime);
        _sTmp                     := Tc2_Standard.CONCAT(_sTmp, _sTab);
        _sTmp                     := Tc2_Standard.CONCAT(_sTmp, Device_To_String(_aWriteList[_iCount].eDevice));
        _sTmp                     := Tc2_Standard.CONCAT(_sTmp, _sTab);
        _sTmp                     := Tc2_Standard.CONCAT(_sTmp, TO_STRING(_aWriteList[_iCount].eSubdevice));
        _sTmp                     := Tc2_Standard.CONCAT(_sTmp, _sTab);
        _sTmp                     := Tc2_Standard.CONCAT(_sTmp, TO_STRING(_aWriteList[_iCount].iErrorNumber));
        _sTmp                     := Tc2_Standard.CONCAT(_sTmp, _sTab);
        _sTmp                     := Tc2_Standard.CONCAT(_sTmp, _aWriteList[_iCount].sText);
        _sTmp                     := Tc2_Standard.CONCAT(_sTmp, _sNewLine);
        Builder(ADR(_sTmp), ADR(_sWriteData), StringLen(ADR(_sTmp)));
      END_IF
      _iCount                     := _iCount + 1;
  END_CASE
  CASE _eFlow
  OF
    E_MESSAGE_FLOW.MSG_FLOW_LINE_CHECK:
    IF NOT (_iCount > _iEnd)
    THEN
      _eFlow                      := E_MESSAGE_FLOW.MSG_FLOW_LINE_BUILD;
    ELSE
      _eState                     := E_PROGRESS.PROGRESS_WORKING;
      _eFlow                      := E_MESSAGE_FLOW.MSG_FLOW_WRITE_FILE_BUSY;
    END_IF
  END_CASE
END_CASE
//-----------------------------------------------------------------------------
//-----------------------------------------------------------------------------
CASE _eState
OF
  E_PROGRESS.PROGRESS_WORKING:
  CASE _eFlow
  OF
    E_MESSAGE_FLOW.MSG_FLOW_WRITE_FILE_BUSY:
      _nStringLength              := StringLen(ADR(_sWriteData));
      IF NOT (_nStringLength > 1)
      THEN
        _eState                   := E_PROGRESS.PROGRESS_DONE; 
       _eFlow                     := E_MESSAGE_FLOW.MSG_FLOW_WRITE_FILE_DONE;
      ELSE
        _eFlow                    := E_MESSAGE_FLOW.MSG_FLOW_WRITE_FILE_END;
        _eRes                     := WriteData(FALSE);
      END_IF
  END_CASE
  CASE _eFlow
  OF
    E_MESSAGE_FLOW.MSG_FLOW_WRITE_FILE_END:
      _eRes                       := WriteData(TRUE);

      IF (_eRes = E_PROGRESS.PROGRESS_ERROR)
      THEN
        _eState                   := E_PROGRESS.PROGRESS_ERROR;

      ELSIF (_eRes = E_PROGRESS.PROGRESS_DONE)
      THEN
        _eState                   := E_PROGRESS.PROGRESS_DONE;
        _eFlow                    := E_MESSAGE_FLOW.MSG_FLOW_WRITE_FILE_DONE;
        _eRes                     := WriteData(FALSE);
      END_IF
  END_CASE
END_CASE
//-----------------------------------------------------------------------------
//-----------------------------------------------------------------------------

BuildFileData                     := _eState;
END_METHOD

METHOD BuildFolder : e_progress
VAR_INPUT
  Execute           : BOOL;
END_VAR
VAR_INST
  _nErrorId   : UDINT;
  _eState     : E_PROGRESS;
  _eFlow      : E_MESSAGE_FLOW;
END_VAR
//-----------------------------------------------------------------------------
IF NOT Execute 
THEN 
	_eState                       := E_PROGRESS.PROGRESS_INIT; 
END_IF 
//-----------------------------------------------------------------------------
IF NOT Check() 
THEN 
	BuildFolder                   := E_PROGRESS.PROGRESS_ERROR; 
	RETURN; 
END_IF
//-----------------------------------------------------------------------------
//-----------------------------------------------------------------------------
CASE _eState
OF
  E_PROGRESS.PROGRESS_INIT:
    IF Execute
    THEN
      _nErrorId                 := 0;
      _bFileCreated             := FALSE;

      _sFolderDate              := FolderDate(_dtLocalTime);
      _eState                   := E_PROGRESS.PROGRESS_BUSY;
      _eFlow                    := E_MESSAGE_FLOW.MSG_FLOW_ROOT;
    END_IF
END_CASE
//-----------------------------------------------------------------------------
//-----------------------------------------------------------------------------
CASE _eState
OF
  E_PROGRESS.PROGRESS_BUSY:
  CASE _eFlow
  OF
    E_MESSAGE_FLOW.MSG_FLOW_ROOT:
      _eFlow                    := E_MESSAGE_FLOW.MSG_FLOW_ROOT_CREATE;
      _fbCreateDir.sPathName    := left(_pDirRoot^,len(_pDirRoot^)-1);
      _fbCreateDir(
              bExecute	        := FALSE);
    
    E_MESSAGE_FLOW.MSG_FLOW_ROOT_CREATE:
      (* create root folder *)
      _fbCreateDir(
              bExecute	        := TRUE);
      IF _fbCreateDir.bBusy
      THEN
        _eFlow                  := E_MESSAGE_FLOW.MSG_FLOW_ROOT_CREATE_BUSY;
      END_IF
    
    E_MESSAGE_FLOW.MSG_FLOW_ROOT_CREATE_BUSY:
      _fbCreateDir(
              bExecute	        := TRUE);
      IF NOT _fbCreateDir.bBusy
      THEN
        _eState                 := E_PROGRESS.PROGRESS_PREPARE;
        _eFlow                  := E_MESSAGE_FLOW.MSG_FLOW_FOLDER;
      END_IF
  END_CASE
END_CASE
//-----------------------------------------------------------------------------
//-----------------------------------------------------------------------------
CASE _eState
OF
  E_PROGRESS.PROGRESS_PREPARE:
  CASE _eFlow
  OF
    E_MESSAGE_FLOW.MSG_FLOW_FOLDER:
      _eFlow                    := E_MESSAGE_FLOW.MSG_FLOW_FOLDER_CREATE;
      _sFolderDate              := FolderDate(_dtLocalTime);
      _fbCreateDir.sPathName    := concat(_pDirRoot^, _sFolderDate);
      _fbCreateDir(
              bExecute	        := FALSE);
  
    E_MESSAGE_FLOW.MSG_FLOW_FOLDER_CREATE:
      (* create active folder *)
      _fbCreateDir(
              bExecute	        := TRUE);
      IF _fbCreateDir.bBusy
      THEN
        _eFlow                  := E_MESSAGE_FLOW.MSG_FLOW_FOLDER_CREATE_BUSY;
      END_IF
    
    E_MESSAGE_FLOW.MSG_FLOW_FOLDER_CREATE_BUSY:
      _fbCreateDir(
              bExecute	        := TRUE);
      IF NOT _fbCreateDir.bBusy
      THEN
        _eState                 := E_PROGRESS.PROGRESS_CHECK;
        _eFlow                  := E_MESSAGE_FLOW.MSG_FLOW_FILE_CREATE_DONE;
        _fbCreateDir(
                bExecute	      := FALSE);
      END_IF
  END_CASE
END_CASE
//-----------------------------------------------------------------------------
//-----------------------------------------------------------------------------
CASE _eState
OF
  E_PROGRESS.PROGRESS_CHECK:
  CASE _eFlow
  OF
    E_MESSAGE_FLOW.MSG_FLOW_FILE_CREATE_DONE:
      _eState                   := E_PROGRESS.PROGRESS_DONE;
      _bFileCreated             := TRUE;

      // build complete file path
      _sTmp                     := concat(concat(_pFileRoot^, _sFolderDate),'.txt');
      _sTmp                     := concat('\', _sTmp);
      _sFilename                := concat(_fbCreateDir.sPathName, _sTmp);
  END_CASE
END_CASE

BuildFolder                     := _eState;
END_METHOD

METHOD Check : BOOL
VAR_INPUT
END_VAR

IF NOT __ISVALIDREF(_stCtrl)
THEN
  _eCheck       := E_MESSAGE_CHECK.POINTER_CTRL_INVALID;
  RETURN;
END_IF

IF NOT __ISVALIDREF(_stState)
THEN
  _eCheck       := E_MESSAGE_CHECK.POINTER_STATE_INVALID;
  RETURN;
END_IF
//-----------------------------------------------------------------
//-----------------------------------------------------------------
IF NOT (_dtLocalTime <> 0)
THEN
  _eCheck       := E_MESSAGE_CHECK.POINTER_TIME_INVALID;
  RETURN;
END_IF

IF NOT (_pMsgList <> 0)
THEN
  _eCheck       := E_MESSAGE_CHECK.POINTER_LIST_INVALID;
  RETURN;
END_IF

IF NOT (_pFileRoot <> 0)
THEN
  _eCheck       := E_MESSAGE_CHECK.POINTER_ROOT_FILE_INVALID;
  RETURN;
END_IF

IF NOT (_pDirRoot <> 0)
THEN
  _eCheck       := E_MESSAGE_CHECK.POINTER_ROOT_DIR_INVALID;
  RETURN;
END_IF

IF NOT __ISVALIDREF(_nMsgIndex)
THEN
  _eCheck       := E_MESSAGE_CHECK.POINTER_MSG_IDX_INVALID;
  RETURN;
END_IF

IF NOT __ISVALIDREF(_nErrIndex)
THEN
  _eCheck       := E_MESSAGE_CHECK.POINTER_ERR_IDX_INVALID;
  RETURN;
END_IF


_eCheck         := E_MESSAGE_CHECK.CHECK_DONE;
Check           := TRUE;
END_METHOD

METHOD Cmd : e_message_state
VAR_INPUT
  Command     : e_message_ctrl;
END_VAR


CASE Command
OF
  E_MESSAGE_CTRL.MSG_CTRL_NULL:
    _eResult                    := E_PROGRESS.PROGRESS_INVALID;
    Cmd                         := E_MESSAGE_STATE.MSG_STATE_NULL;

  E_MESSAGE_CTRL.MSG_CTRL_INIT:
    _eResult                    := BuildFolder(FALSE);
    Cmd                         := E_MESSAGE_STATE.MSG_STATE_INIT;

  E_MESSAGE_CTRL.MSG_CTRL_IDLE:
    _eResult                    := BuildFileData(FALSE);
    Cmd                         := E_MESSAGE_STATE.MSG_STATE_IDLE;

  E_MESSAGE_CTRL.MSG_CTRL_WRITE:
    _eResult                    := BuildFileData(FALSE);
    Cmd                         := E_MESSAGE_STATE.MSG_STATE_WRITE;
    IF (_nMsgIndex = 0)
    THEN
       // go back to sleep
      _eResult                := E_PROGRESS.PROGRESS_DONE;
    END_IF
ELSE
    //_eResult                    := E_PROGRESS.PROGRESS_ERROR;
    Cmd                         := E_MESSAGE_STATE.MSG_STATE_NULL;
END_CASE
END_METHOD

PROPERTY Ctrl : REFERENCE to ST_MESSAGE_CTRL
SET
_stCtrl ref= Ctrl;
END_SET
END_PROPERTY

PROPERTY FileCreated : bool
GET
FileCreated := _bFileCreated;
END_GET
END_PROPERTY

PROPERTY State : REFERENCE TO ST_MESSAGE_STATE
SET
_stState ref= State;
END_SET
END_PROPERTY

END_FUNCTION_BLOCK

// ---- _MSG/class/fb_MessageData.TcPOU
FUNCTION_BLOCK ABSTRACT fb_MessageData IMPLEMENTS I_MessageData
VAR CONSTANT
{attribute 'hide'}
  STR_LEN       : UDINT := 524_288;
END_VAR
VAR
  _eCheck       : E_MESSAGE_CHECK;            // pointer check state

  _pFileRoot    : POINTER TO STRING(255);     // you decide (example in GVL_MSG.LOG_FILE)
  _pDirRoot     : POINTER TO STRING(255);     // see GVL_MSG.LOG_DIR

  _nMsgIndex    : REFERENCE TO UINT;          // Hypnos IS the only one in the village, if there are more you need more villages
  _nErrIndex    : REFERENCE TO UINT;          // Thanatos, Hypnos stern and more serious brother

  _dtLocalTime  : POINTER TO DT;
  _pMsgList     : POINTER TO ARRAY[1..GVL_MSG_XTS.MAX_MESSAGE] OF ST_Message; // attach your list here

	_rtrigReset   : Tc2_Standard.R_TRIG;
	_aWriteList   : ARRAY[1..GVL_MSG_XTS.MAX_MESSAGE] OF ST_Message;
	_sWriteData   : STRING(STR_LEN);
	_sNewLine     : STRING := '$N';
	_sTab         : STRING := '$T';
	_iCount, 
	_iStart, 
	_iEnd         : UINT;

	_fbCreateDir  : Tc2_System.FB_CreateDir;
	_sTmp         : STRING(256);
	_sFilename    : STRING(256);
	_sFolderDate  : STRING;
	_bFileCreated : BOOL;

	_fbFileOpen   : Tc2_System.FB_FileOpen;
	_fbFileWrite  : Tc2_System.FB_FileWrite;
	_fbFileClose  : Tc2_System.FB_FileClose;
END_VAR

METHOD Builder : BOOL // string concat for length > 255
VAR_INPUT
  pInString   : POINTER TO STRING;
  pOutString  : POINTER TO STRING(STR_LEN);
  Length      : UINT;
END_VAR
VAR
  Counter     : UDINT;
  pInWork     : POINTER TO BYTE;
  pOutWork    : POINTER TO BYTE;
END_VAR
pOutWork := pOutString;
pInWork := pInString;
Counter := 0;

(*check termination*)
WHILE (pOutWork^ <> 0) AND
      (Counter < STR_LEN+1)
DO
  Counter := Counter + 1;
  pOutWork := pOutWork + 1;
END_WHILE

(* append only if data fits into output *)
IF (Counter + Length < STR_LEN+1)
THEN

  (* append data *)
  FOR Counter := 1 TO Length
  DO
    pOutWork^ := pInWork^;
    pOutWork := pOutWork + 1;
    pInWork := pInWork + 1;
  END_FOR

  (* terminate *)
  pOutWork := pOutWork + 1;
  pOutWork^ := 0;
END_IF
END_METHOD

METHOD Check : BOOL
VAR_INPUT
END_VAR

IF NOT (_dtLocalTime <> 0)
THEN
  _eCheck       := E_MESSAGE_CHECK.POINTER_TIME_INVALID;
  RETURN;
END_IF

IF NOT (_pMsgList <> 0)
THEN
  _eCheck       := E_MESSAGE_CHECK.POINTER_LIST_INVALID;
  RETURN;
END_IF

IF NOT (_pFileRoot <> 0)
THEN
  _eCheck       := E_MESSAGE_CHECK.POINTER_ROOT_FILE_INVALID;
  RETURN;
END_IF

IF NOT (_pDirRoot <> 0)
THEN
  _eCheck       := E_MESSAGE_CHECK.POINTER_ROOT_DIR_INVALID;
  RETURN;
END_IF

IF NOT __ISVALIDREF(_nMsgIndex)
THEN
  _eCheck       := E_MESSAGE_CHECK.POINTER_MSG_IDX_INVALID;
  RETURN;
END_IF

IF NOT __ISVALIDREF(_nErrIndex)
THEN
  _eCheck       := E_MESSAGE_CHECK.POINTER_ERR_IDX_INVALID;
  RETURN;
END_IF


_eCheck         := E_MESSAGE_CHECK.CHECK_DONE;
Check           := TRUE;
END_METHOD

METHOD Device_to_String : string
VAR_INPUT
  eMsgDevice    : e_Device;
END_VAR
VAR
  sId                 : STRING := '_ID_';
  nId                 : UDINT;
END_VAR
IF (eMsgDevice < e_device.General)
THEN
  // below general case
  nId := TO_UDINT(eMsgDevice);
  //sId := concat(sId, TO_STRING(nId));

  //Device_to_String := concat(TO_STRING(eMsgDevice), sId);
  Device_to_String := TO_STRING(eMsgDevice);

ELSE
  IF (eMsgDevice >= e_Device.DataProduct)
  THEN
    nId := eMsgDevice MOD e_Device.DataProduct;
    sId := concat(sId, TO_STRING(nId));
 
    Device_to_String := concat(TO_STRING(e_Device.DataProduct), sId);

  ELSIF (eMsgDevice >= e_Device.Application)
  THEN
    nId := eMsgDevice MOD e_Device.Application;
    sId := concat(sId, TO_STRING(nId));
 
    Device_to_String := concat(TO_STRING(e_Device.Application), sId);

  ELSIF (eMsgDevice >= e_Device.TicketListCtrl)
  THEN
    nId := eMsgDevice MOD e_Device.TicketListCtrl;
    sId := concat(sId, TO_STRING(nId));
 
    Device_to_String := concat(TO_STRING(e_Device.TicketListCtrl), sId);

  ELSIF (eMsgDevice >= e_Device.ProcessListCtrl)
  THEN
    nId := eMsgDevice MOD e_Device.ProcessListCtrl;
    sId := concat(sId, TO_STRING(nId));
 
    Device_to_String := concat(TO_STRING(e_Device.ProcessListCtrl), sId);

  ELSIF (eMsgDevice >= e_Device.Process)
  THEN
    nId := eMsgDevice MOD e_Device.Process;
    sId := concat(sId, TO_STRING(nId));
 
    Device_to_String := concat(TO_STRING(e_Device.Process), sId);

  ELSIF (eMsgDevice >= e_Device.MetricsAxis)
  THEN
    nId := eMsgDevice MOD e_Device.MetricsAxis;
    sId := concat(sId, TO_STRING(nId));
 
    Device_to_String := concat(TO_STRING(e_device.MetricsAxis), sId);

  ELSIF (eMsgDevice >= e_Device.MetricsXts)
  THEN
    nId := eMsgDevice MOD e_Device.MetricsXts;
    sId := concat(sId, TO_STRING(nId));
 
    Device_to_String := concat(TO_STRING(e_device.MetricsXts), sId);

  ELSIF (eMsgDevice >= e_device.XfcAxis)
  THEN
    nId := eMsgDevice MOD e_device.XfcAxis;
    sId := concat(sId, TO_STRING(nId));
 
    Device_to_String := concat(TO_STRING(e_device.XfcAxis), sId);

  ELSIF (eMsgDevice >= e_device.Axis)
  THEN
    nId := eMsgDevice MOD e_device.Axis;
    sId := concat(sId, TO_STRING(nId));
 
    Device_to_String := concat(TO_STRING(e_device.Axis), sId);

  ELSIF (eMsgDevice >= e_device.NciChannelCtrl)
  THEN
    nId := eMsgDevice MOD e_device.NciChannelCtrl;
    sId := concat(sId, TO_STRING(nId));
 
    Device_to_String := concat(TO_STRING(e_device.NciChannelCtrl), sId);

  ELSIF (eMsgDevice >= e_device.NciChannel)
  THEN
    nId := eMsgDevice MOD e_device.NciChannel;
    sId := concat(sId, TO_STRING(nId));
 
    Device_to_String := concat(TO_STRING(e_device.NciChannel), sId);

  ELSIF (eMsgDevice >= e_Device.Camming)
  THEN
    nId := eMsgDevice MOD e_Device.Camming;
    sId := concat(sId, TO_STRING(nId));
 
    Device_to_String := concat(TO_STRING(e_device.Camming), sId);

  ELSIF (eMsgDevice >= e_Device.XtsStation)
  THEN
    nId := eMsgDevice MOD e_Device.XtsStation;
    sId := concat(sId, TO_STRING(nId));
 
    Device_to_String := concat(TO_STRING(e_device.XtsStation), sId);

  ELSIF (eMsgDevice >= e_Device.XfcTouchProbe)
  THEN
    nId := eMsgDevice MOD e_Device.XfcTouchProbe;
    sId := concat(sId, TO_STRING(nId));
 
    Device_to_String := concat(TO_STRING(e_device.XfcTouchProbe), sId);

  ELSIF (eMsgDevice >= e_Device.XfcTriggerBox)
  THEN
    nId := eMsgDevice MOD e_Device.XfcTriggerBox;
    sId := concat(sId, TO_STRING(nId));
 
    Device_to_String := concat(TO_STRING(e_device.XfcTriggerBox), sId);

  ELSIF (eMsgDevice >= e_Device.XtsTransportUnit)
  THEN
    nId := eMsgDevice MOD e_Device.XtsTransportUnit;
    sId := concat(sId, TO_STRING(nId));
 
    Device_to_String := concat(TO_STRING(e_device.XtsTransportUnit), sId);

  ELSIF (eMsgDevice >= e_Device.MoverCtrl)
  THEN
    nId := eMsgDevice MOD e_Device.MoverCtrl;
    sId := concat(sId, TO_STRING(nId));
 
    Device_to_String := concat(TO_STRING(e_device.MoverCtrl), sId);

  ELSIF (eMsgDevice >= e_Device.Mover)
  THEN
    nId := eMsgDevice MOD e_Device.Mover;
    sId := concat(sId, TO_STRING(nId));
 
    Device_to_String := concat(TO_STRING(e_device.Mover), sId);

  ELSIF (eMsgDevice >= e_Device.XpuCtrl)
  THEN
    nId := eMsgDevice MOD e_Device.XpuCtrl;
    sId := concat(sId, TO_STRING(nId));
 
    Device_to_String := concat(TO_STRING(e_device.XpuCtrl), sId);

  ELSIF (eMsgDevice >= e_Device.Xpu)
  THEN
    nId := eMsgDevice MOD e_Device.Xpu;
    sId := concat(sId, TO_STRING(nId));
 
    Device_to_String := concat(TO_STRING(e_device.Xpu), sId);

  ELSIF (eMsgDevice >= e_Device.CaGroup)
  THEN
    nId := eMsgDevice MOD e_Device.CaGroup;
    sId := concat(sId, TO_STRING(nId));
 
    Device_to_String := concat(TO_STRING(e_device.CaGroup), sId);

  ELSIF (eMsgDevice >= e_Device.General)
  THEN
    nId := eMsgDevice MOD e_Device.General;
    //sId := concat(sId, TO_STRING(nId));
 
    Device_to_String := TO_STRING(e_device.General);

  ELSE
    Device_to_String := TO_STRING(eMsgDevice);
  END_IF
END_IF
END_METHOD

PROPERTY DirRoot : POINTER to string(255)
SET
_pDirRoot := DirRoot;
END_SET
END_PROPERTY

PROPERTY ErrorIndex : reference to uint
SET
_nErrIndex  REF= ErrorIndex;
END_SET
END_PROPERTY

PROPERTY FileRoot : pointer to string(255)
SET
_pFileRoot := FileRoot;
END_SET
END_PROPERTY

METHOD FolderDate : STRING
VAR_INPUT
	LocalTime   : POINTER TO DT;
END_VAR
VAR
	sTmp        : STRING;
END_VAR
IF NOT (LocalTime <> 0)
THEN
	FolderDate := 'NULL';
	RETURN;
END_IF

sTmp := DT_TO_STRING(LocalTime^);

// cut off #dt literal
sTmp := right(sTmp, len(sTmp)-3);

sTmp := replace(sTmp, '_', 1, 5);
sTmp := replace(sTmp, '_', 1, 8);

sTmp := left(sTmp,10);	// year_month_day

FolderDate := sTmp;
END_METHOD

PROPERTY LocalTime : pointer to DT
SET
_dtLocalTime := LocalTime;
END_SET
END_PROPERTY

PROPERTY MessageIndex : reference to uint
SET
_nMsgIndex   REF= MessageIndex;
END_SET
END_PROPERTY

PROPERTY MsgList : pointer to ARRAY[1..GVL_MSG_XTS.MAX_MESSAGE] OF st_message
SET
_pMsgList := MsgList;
END_SET
END_PROPERTY

METHOD StringLen : UINT // 	string length for len > 255
VAR_INPUT
  pInString		: POINTER TO STRING(STR_LEN);
END_VAR
VAR
	Counter			: UINT;
	pInWork			: POINTER TO BYTE;
END_VAR
pInWork := pInString;
Counter := 0;

WHILE (pInWork^ <> 0) AND
			(Counter < STR_LEN)
DO
	Counter := Counter + 1;
	pInWork := pInWork + 1;
END_WHILE

StringLen := Counter;
END_METHOD

METHOD WriteData  : e_progress
VAR_INPUT
  bExecute        : BOOL;
END_VAR
VAR_INST
  _eState         : e_progress;
  _bError         : BOOL;
  _nErrorId       : UDINT;
END_VAR
IF NOT bExecute
THEN
  _eState                     := E_PROGRESS.PROGRESS_INIT;
END_IF

CASE _eState 
OF

	E_PROGRESS.PROGRESS_INIT:
    _fbFileOpen(
        sPathName             := _sFilename, 
        nMode                 := FOPEN_MODEAPPEND OR FOPEN_MODEPLUS, 
        ePath                 := PATH_GENERIC, 
        bExecute              := FALSE, 
        tTimeout              := T#5S);

    _fbFileWrite(
        hFile                 := _fbFileOpen.hFile, 
        pWriteBuff            := ADR(_sWriteData), 
        cbWriteLen            := StringLen(ADR(_sWriteData)),
        bExecute              := FALSE, 
        tTimeout              := T#5S);

    _fbFileClose(
        hFile                 := _fbFileOpen.hFile, 
        bExecute              := FALSE, 
        tTimeout              := T#5S);


		IF bExecute
		THEN
      _nErrorId               := 0;
      _eState                 := E_PROGRESS.PROGRESS_BUSY;
		END_IF

	E_PROGRESS.PROGRESS_BUSY:
		_fbFileOpen(bExecute      := TRUE);

    IF _fbFileOpen.bError
    THEN
      _nErrorId               := _fbFileOpen.nErrId;
      _eState                 := E_PROGRESS.PROGRESS_ERROR;

		ELSIF _fbFileOpen.bBusy
		THEN
      _eState                 := E_PROGRESS.PROGRESS_PREPARE;
		END_IF

	E_PROGRESS.PROGRESS_PREPARE:
		_fbFileOpen(bExecute      := TRUE);
		IF NOT _fbFileOpen.bBusy
		THEN
		  _fbFileOpen(bExecute    := FALSE);
      _eState                 := E_PROGRESS.PROGRESS_STARTUP;
		END_IF

	E_PROGRESS.PROGRESS_STARTUP:
    _fbFileWrite(
        hFile                 := _fbFileOpen.hFile, 
        pWriteBuff            := ADR(_sWriteData), 
        cbWriteLen            := StringLen(ADR(_sWriteData)),
        bExecute              := TRUE, 
        tTimeout              := T#5S);

    IF _fbFileWrite.bError
    THEN
      _nErrorId               := _fbFileWrite.nErrId;
      _eState                 := E_PROGRESS.PROGRESS_ERROR;

		ELSIF _fbFileWrite.bBusy
		THEN
      _eState                 := E_PROGRESS.PROGRESS_CHECK;
		END_IF

	E_PROGRESS.PROGRESS_CHECK:
	  _fbFileWrite(bExecute     := TRUE);
		IF NOT _fbFileWrite.bBusy
		THEN
			_fbFileWrite(bExecute   := FALSE);
      _eState                 := E_PROGRESS.PROGRESS_OCCUPIED;
		END_IF

	E_PROGRESS.PROGRESS_OCCUPIED:
    _fbFileClose(
        hFile                 := _fbFileOpen.hFile, 
        bExecute              := TRUE, 
        tTimeout              := T#5S);

    IF _fbFileClose.bError
    THEN
      _nErrorId               := _fbFileClose.nErrId;
      _eState                 := E_PROGRESS.PROGRESS_ERROR;

		ELSIF _fbFileClose.bBusy
		THEN
      _eState                 := E_PROGRESS.PROGRESS_WORKING;
		END_IF

	E_PROGRESS.PROGRESS_WORKING:
    _fbFileClose(bExecute     := TRUE);
		IF NOT _fbFileClose.bBusy
		THEN
			_fbFileClose(bExecute   := FALSE);
      _eState                 := E_PROGRESS.PROGRESS_DONE;
		END_IF

END_CASE
CASE _eState
OF
  E_PROGRESS.PROGRESS_ERROR:
		_fbFileOpen (bExecute     := FALSE);
    _fbFileWrite(bExecute     := FALSE);
    _fbFileClose(bExecute     := FALSE);


END_CASE




WriteData                     := _eState;
END_METHOD

END_FUNCTION_BLOCK

// ---- _MSG/class/fb_LocalTime.TcPOU
//-----------------------------------------------------------------------------------------------
//
//  As time goes by...
//
//  HAUD 2026 07 23
//  - timezone to match UTC device time.
//-----------------------------------------------------------------------------------------------
FUNCTION_BLOCK fb_LocalTime
VAR
  _eState                 : e_progress;   // self startup state, reaches WORKING when done.
  _stSystemtime           : Tc2_Utilities.TIMESTRUCT;

  _stUtcTime              : Tc2_Utilities.T_FILETIME64; // CPU time as 64bit ULINT, meant to be used for measurement
  _sUtcTime               : STRING;
  _dtUtcTime              : DT;

  _stLocalTime            : Tc2_Utilities.T_FILETIME64; // In every wood, in every spring,there is a different green.
  _sLocalTime             : STRING;
  _dtLocalTime            : DT;

  _eTimeZoneId            : Tc2_Utilities.E_TimeZoneID;
  _stTimeZoneInfo         : Tc2_Utilities.ST_TimeZoneInformation;
  _fbGetTimeZoneInfo      : Tc2_Utilities.FB_GetTimeZoneInformation;
  _fbFileTimeToLocalTime  : Tc2_Utilities.FB_FileTime64ToTzSpecificLocalTime;
  _nErrorId               : UDINT;
  _bError                 : BOOL;
END_VAR

//-----------------------------------------------------------------------------------------------
// infosys: https://infosys.beckhoff.com/english.php?content=../content/1033/tcplclib_tc2_system/3622991755.html&id=6591934602709167291
//-----------------------------------------------------------------------------------------------
// This function can be used to read the operating system timestamp. 
// The timestamp is a 64-bit integer value, with an accuracy of 100 ns, 
// which is updated with every call of the PLC. 
// Among other things, it can be used for timing tasks or time measurements. 
// One unit corresponds to 100 ns. 
// The time represents the number of 100 ns intervals since January 1, 1601 (UTC).
//-----------------------------------------------------------------------------------------------
//-----------------------------------------------------------------------------------------------
_stUtcTime                      := F_GetSystemTime(); // UTC time, no delay --> CPU time direct
//-----------------------------------------------------------------------------------------------
//-----------------------------------------------------------------------------------------------
// build UTC time
_sUtcTime                       := SYSTEMTIME_TO_STRING( FILETIME64_TO_SYSTEMTIME( _stUtcTime ));
_dtUtcTime                      := systemtime_to_dt    ( FILETIME64_TO_SYSTEMTIME( _stUtcTime ));
//-----------------------------------------------------------------------------------------------
//-----------------------------------------------------------------------------------------------
// state machine for getting timezone information and add the offset to UTC time
//-----------------------------------------------------------------------------------------------
CASE _eState
OF
  E_PROGRESS.PROGRESS_INVALID:
    _eState                     := E_PROGRESS.PROGRESS_INIT;
    _fbGetTimeZoneInfo(
                      sNetID    := '', 
                      bExecute  := FALSE,
                      bError    => _bError,
                      nErrID    => _nErrorId, 
                      tzID      => _eTimeZoneId, 
                      tzInfo    => _stTimeZoneInfo);
END_CASE
//---------------------------------------------------------------------------------------------
//---------------------------------------------------------------------------------------------
CASE _eState
OF
  E_PROGRESS.PROGRESS_INIT:
    _fbGetTimeZoneInfo(
                      sNetID    := '', 
                      bExecute  := TRUE,
                      bError    => _bError,
                      nErrID    => _nErrorId, 
                      tzID      => _eTimeZoneId, 
                      tzInfo    => _stTimeZoneInfo);

    IF (_fbGetTimeZoneInfo.bBusy)
    THEN
      _eState                   := E_PROGRESS.PROGRESS_PREPARE;
    END_IF
END_CASE
//---------------------------------------------------------------------------------------------
//---------------------------------------------------------------------------------------------
CASE _eState
OF
  E_PROGRESS.PROGRESS_PREPARE:
    _fbGetTimeZoneInfo(
                      sNetID    := '', 
                      bExecute  := TRUE,
                      bError    => _bError,
                      nErrID    => _nErrorId, 
                      tzID      => _eTimeZoneId, 
                      tzInfo    => _stTimeZoneInfo);

    IF NOT (_fbGetTimeZoneInfo.bBusy)
    THEN
      _fbGetTimeZoneInfo(
                      sNetID    := '', 
                      bExecute  := FALSE);

      _eState                   := E_PROGRESS.PROGRESS_WORKING;
    END_IF
END_CASE
//---------------------------------------------------------------------------------------------
//---------------------------------------------------------------------------------------------
CASE _eState
OF
  E_PROGRESS.PROGRESS_WORKING:
    _fbFileTimeToLocalTime(
                      in        := _stUtcTime, 
                      tzInfo    := _stTimeZoneInfo, 
                      out       => _stLocalTime, 
                      eTzID     => _eTimeZoneId);

  // build local time
  _stSystemtime                 := FILETIME64_TO_SYSTEMTIME( _stLocalTime );
  _sLocalTime                   := SYSTEMTIME_TO_STRING    ( _stSystemtime );
  _dtLocalTime                  := systemtime_to_dt        ( _stSystemtime );


  IF (_stSystemtime.wHour   = 0) AND
     (_stSystemtime.wMinute = 0) AND
     (_stSystemtime.wSecond = 0)
  THEN
    //  The passing seasons are but ripples ever repeated in the long long stream.
    _eState                     := E_PROGRESS.PROGRESS_INIT;
  END_IF
END_CASE
//---------------------------------------------------------------------------------------------
//---------------------------------------------------------------------------------------------

METHOD FolderDate : STRING
VAR_INPUT
	LocalTime   : POINTER TO DT;
END_VAR
VAR
	sTmp        : STRING;
END_VAR
IF NOT (LocalTime <> 0)
THEN
	FolderDate := 'NULL';
	RETURN;
END_IF

sTmp := DT_TO_STRING(LocalTime^);

// cut off #dt literal
sTmp := right(sTmp, len(sTmp)-3);

sTmp := replace(sTmp, '_', 1, 5);
sTmp := replace(sTmp, '_', 1, 8);

sTmp := left(sTmp,10);	// year_month_day

FolderDate := sTmp;
END_METHOD

PROPERTY LocalTime : DT
GET
LocalTime := _dtLocalTime;
END_GET
END_PROPERTY

PROPERTY LocalTimeString : string
GET
IF (len(_sLocalTime) >1)
THEN
  LocalTimeString := _sLocalTime;
ELSE
  LocalTimeString := _sUtcTime;
END_IF
END_GET
END_PROPERTY

PROPERTY State : e_progress
GET
State := _eState;
END_GET
END_PROPERTY

PROPERTY UtcTime : DT
GET
UtcTime := _dtUtcTime;
END_GET
END_PROPERTY

PROPERTY UtcTimeString : string
GET
UtcTimeString := _sUtcTime;
END_GET
END_PROPERTY

END_FUNCTION_BLOCK

// ---- APPLICATION/MAIN_APP.TcPOU
//---------------------------------------------------------------------------------------------------------------
//
//  HAUD 2026.01.16
//
//  - ExternControl
//
//    - cyclic call to simulation class which handshakes the XtsStations in XtsTransport PLC
//
//---------------------------------------------------------------------------------------------------------------
PROGRAM MAIN_APP
VAR
  eInitXtsTransport   AT %I*    : e_progress;
  eInit                         : E_PROGRESS;   // application startup state info

  nProcess          : UINT;

  bNext             : BOOL := TRUE;
  bEnter            : BOOL := TRUE;
  bLeave            : BOOL := TRUE;

  tProcess          : ARRAY[1..MAX_PROCESS] OF TIME;

  eMtrState,
  eMsgState         : E_MESSAGE_STATE;
  eMtrProgress,
  eMsgProgress      : e_progress;
  stMsg             : ST_Message;
  //-------------------------------------------------------------------------------------------------------------
  tIdleWriteApplication   : TIME := T#5S;
  tIdleWriteMetric        : TIME := T#5S;
  tonIdleWriteApplication : Tc2_Standard.TON;
  tonIdleWriteMetric      : Tc2_Standard.TON;
  //-------------------------------------------------------------------------------------------------------------
END_VAR

//#################################################################################################################
// Local time; used for timestamps
//#################################################################################################################
GVL_MSG_XTS.fbLocalTime();
GVL_MSG_XTS.sLocalTime                                      := GVL_MSG_XTS.fbLocalTime.LocalTimeString;
GVL_MSG_XTS.dtLocalTime                                     := GVL_MSG_XTS.fbLocalTime.LocalTime;
//#################################################################################################################
//#################################################################################################################
//-----------------------------------------------------------------------------------------------------------------
//-----------------------------------------------------------------------------------------------------------------
// check for MAIN.eInit
//  - wait for fb_TransportUnit to be fully started up
//-----------------------------------------------------------------------------------------------------------------
IF NOT (eInitXtsTransport = E_PROGRESS.PROGRESS_DONE) THEN eInit   := E_PROGRESS.PROGRESS_INVALID; RETURN; END_IF
//-----------------------------------------------------------------------------------------------------------------
//-----------------------------------------------------------------------------------------------------------------
//-----------------------------------------------------------------------------------------------------------------
// /assign dataflow
//-----------------------------------------------------------------------------------------------------------------
FOR nProcess := 1 TO MAX_PROCESS
DO
  GVL_APPLICATION.Simulation[nProcess].ProcessId            := nProcess;
  GVL_APPLICATION.Simulation[nProcess].StationCtrl          := ADR(GVL_XTS.StationCtrl);
  GVL_APPLICATION.Simulation[nProcess].StationState         := ADR(GVL_XTS.StationState);

  GVL_APPLICATION.Simulation[nProcess].ProcessTime          := tProcess[nProcess];
  GVL_APPLICATION.Simulation[nProcess].MessageLevel         := GVL_MSG_XTS.MessageLevel;
END_FOR
//-----------------------------------------------------------------------------------------------------------------
//-----------------------------------------------------------------------------------------------------------------
Init();
//-----------------------------------------------------------------------------------------------------------------
//-----------------------------------------------------------------------------------------------------------------
// react to operation modes
//-----------------------------------------------------------------------------------------------------------------
//-----------------------------------------------------------------------------------------------------------------
CASE GVL_XTS.XtsTransportCtrl.Cmd
OF
  E_XTS_TRANSPORT_CTRL.CMD_INIT,
  E_XTS_TRANSPORT_CTRL.CMD_GROUP_CLEAR:

    FOR nProcess := 1 TO MAX_PROCESS
    DO
      GVL_APPLICATION.Simulation[nProcess].Init(); // clearing of XtsStations and Simulation
    END_FOR
END_CASE

CASE (GVL_XTS.XtsTransportState.State MOD E_PROGRESS.PROGRESS_DONE)
OF
  E_XTS_TRANSPORT_STATE.TRANSPORT_INIT,
  E_XTS_TRANSPORT_STATE.TRANSPORT_GROUP_CLEAR:
    FOR nProcess := 1 TO MAX_PROCESS
    DO
      GVL_APPLICATION.Simulation[nProcess].Disable(); // switch off XtsStations and clear Simulation

      GVL_APPLICATION.Simulation[nProcess].EnableProcess    := 0;
      GVL_APPLICATION.Simulation[nProcess].MoverEnter       := FALSE;
      GVL_APPLICATION.Simulation[nProcess].MoverOut         := FALSE;

      GVL_APPLICATION.Simulation[nProcess].Cycle();
    END_FOR

  E_XTS_TRANSPORT_STATE.TRANSPORT_START,
  E_XTS_TRANSPORT_STATE.TRANSPORT_RESTART:

    FOR nProcess := 1 TO MAX_PROCESS
    DO
      GVL_APPLICATION.Simulation[nProcess].Next(bNext);
      GVL_APPLICATION.Simulation[nProcess].Cycle();
    END_FOR
ELSE
  CASE (GVL_XTS.XtsTransportState.State MOD E_PROGRESS.PROGRESS_WORKING)
  OF
  E_XTS_TRANSPORT_STATE.TRANSPORT_START,
  E_XTS_TRANSPORT_STATE.TRANSPORT_RESTART:
    FOR nProcess := 1 TO MAX_PROCESS
    DO
      IF (GVL_APPLICATION.Simulation[nProcess].StationCount > 0)
      THEN
        GVL_APPLICATION.Simulation[nProcess].EnableProcess  := TO_DWORD(EXPT(2,GVL_APPLICATION.Simulation[nProcess].StationCount))-1;
        GVL_APPLICATION.Simulation[nProcess].MoverEnter     := TRUE;
        GVL_APPLICATION.Simulation[nProcess].MoverOut       := TRUE;

      END_IF

      GVL_APPLICATION.Simulation[nProcess].Next(bNext);
      GVL_APPLICATION.Simulation[nProcess].Cycle();
    END_FOR
  END_CASE
END_CASE
//-----------------------------------------------------------------------------------------------------------------
//-----------------------------------------------------------------------------------------------------------------
//#################################################################################################################
// /logging
//#################################################################################################################
GVL_MSG_XTS.ApplicationMessageData.Ctrl                     REF= GVL_MSG_XTS.ApplicationMessageCtrl;
GVL_MSG_XTS.ApplicationMessageData.State                    REF= GVL_MSG_XTS.ApplicationMessageState;

GVL_MSG_XTS.ApplicationMessageData.MessageIndex             REF= GVL_MSG_XTS.MessageApplicationIndex;
GVL_MSG_XTS.ApplicationMessageData.ErrorIndex               REF= GVL_MSG_XTS.MessageApplicationError;

GVL_MSG_XTS.ApplicationMessageData.DirRoot                  :=   ADR(GVL_MSG_XTS.LOG_DIR);
GVL_MSG_XTS.ApplicationMessageData.FileRoot                 :=   ADR(GVL_MSG_XTS.LOG_FILE_APP);
GVL_MSG_XTS.ApplicationMessageData.MsgList                  :=   ADR(GVL_MSG_XTS.ApplicationMessages);
GVL_MSG_XTS.ApplicationMessageData.LocalTime                :=   ADR(GVL_MSG_XTS.dtLocalTime);

GVL_MSG_XTS.ApplicationMessageData();

eMsgState                                   := f_GetState   (GVL_MSG_XTS.ApplicationMessageState.State);
eMsgProgress                                := f_GetProgress(GVL_MSG_XTS.ApplicationMessageState.State);


CASE eMsgState
OF
  E_MESSAGE_STATE.MSG_STATE_NULL:
    CASE eMsgProgress
    OF
      E_PROGRESS.PROGRESS_INVALID:
        IF (GVL_MSG_XTS.MessageApplicationIndex > GVL_MSG_XTS.MAX_MESSAGE/100) OR
           (GVL_MSG_XTS.MessageApplicationError > 0)
        THEN
          GVL_MSG_XTS.ApplicationMessageCtrl.Cmd            := E_MESSAGE_CTRL.MSG_CTRL_WRITE;
        ELSE
          tonIdleWriteApplication(IN := TRUE, PT:= tIdleWriteApplication);
          IF (tonIdleWriteApplication.Q)
          THEN
            GVL_MSG_XTS.TransportMessageCtrl.Cmd            := E_MESSAGE_CTRL.MSG_CTRL_WRITE;
          END_IF
        END_IF
    END_CASE

  E_MESSAGE_STATE.MSG_STATE_WRITE:
    CASE eMsgProgress
    OF
      E_PROGRESS.PROGRESS_ERROR,
      E_PROGRESS.PROGRESS_DONE:
        tonIdleWriteApplication(IN := FALSE, PT:= tIdleWriteApplication);
        GVL_MSG_XTS.ApplicationMessageCtrl.Cmd              := E_MESSAGE_CTRL.MSG_CTRL_NULL;
    END_CASE

ELSE
    CASE eMsgProgress
    OF
      E_PROGRESS.PROGRESS_DONE:
        GVL_MSG_XTS.ApplicationMessageCtrl.Cmd              := E_MESSAGE_CTRL.MSG_CTRL_NULL;
    END_CASE
END_CASE
//#################################################################################################################
// logging/
//#################################################################################################################
//#################################################################################################################
//  /Transport Metrics
//#################################################################################################################
GVL_MSG_XTS.MetricsMessageData.Ctrl                         REF= GVL_MSG_XTS.MetricsMessageCtrl;
GVL_MSG_XTS.MetricsMessageData.State                        REF= GVL_MSG_XTS.MetricsMessageState;

GVL_MSG_XTS.MetricsMessageData.MessageIndex                 REF= GVL_MSG_XTS.MessageMetricsIndex;
GVL_MSG_XTS.MetricsMessageData.ErrorIndex                   REF= GVL_MSG_XTS.MessageMetricsError;

GVL_MSG_XTS.MetricsMessageData.DirRoot                      :=   ADR(GVL_MSG_XTS.LOG_DIR);
GVL_MSG_XTS.MetricsMessageData.FileRoot                     :=   ADR(GVL_MSG_XTS.LOG_FILE_METRIC);
GVL_MSG_XTS.MetricsMessageData.MsgList                      :=   ADR(GVL_MSG_XTS.MetricsMessages);
GVL_MSG_XTS.MetricsMessageData.LocalTime                    :=   ADR(GVL_MSG_XTS.dtLocalTime);

GVL_MSG_XTS.MetricsMessageData();

eMtrState                                   := f_GetState   (GVL_MSG_XTS.MetricsMessageState.State);
eMtrProgress                                := f_GetProgress(GVL_MSG_XTS.MetricsMessageState.State);

CASE eMtrState
OF
  E_MESSAGE_STATE.MSG_STATE_NULL:
    CASE eMtrProgress
    OF
      E_PROGRESS.PROGRESS_INVALID:
        IF (GVL_MSG_XTS.MessageMetricsIndex > GVL_MSG_XTS.MAX_MESSAGE/100) OR
           (GVL_MSG_XTS.MessageMetricsError > 0)
        THEN
          GVL_MSG_XTS.MetricsMessageCtrl.Cmd                := E_MESSAGE_CTRL.MSG_CTRL_WRITE;
        ELSE
          tonIdleWriteMetric(IN := TRUE, PT:= tIdleWriteMetric);
          IF (tonIdleWriteMetric.Q)
          THEN
            GVL_MSG_XTS.TransportMessageCtrl.Cmd            := E_MESSAGE_CTRL.MSG_CTRL_WRITE;
          END_IF
        END_IF
    END_CASE

  E_MESSAGE_STATE.MSG_STATE_WRITE:
    CASE eMtrProgress
    OF
      E_PROGRESS.PROGRESS_ERROR,
      E_PROGRESS.PROGRESS_DONE:
        tonIdleWriteMetric(IN := FALSE, PT:= tIdleWriteMetric);
        GVL_MSG_XTS.MetricsMessageCtrl.Cmd                  := E_MESSAGE_CTRL.MSG_CTRL_NULL;
    END_CASE
ELSE
    CASE eMtrProgress
    OF
      E_PROGRESS.PROGRESS_DONE:
        GVL_MSG_XTS.MetricsMessageCtrl.Cmd                  := E_MESSAGE_CTRL.MSG_CTRL_NULL;
    END_CASE
END_CASE
//#################################################################################################################
//  Transport Metrics/
//#################################################################################################################
//#################################################################################################################
//#################################################################################################################

ACTION Init:
CASE eInit
OF
  E_PROGRESS.PROGRESS_INVALID:          // startup procedure for your application
    eInit                               := E_PROGRESS.PROGRESS_INIT;


  E_PROGRESS.PROGRESS_INIT:
      nProcess                                        := 1;
      tProcess[nProcess]                              := T#0MS;

      GVL_APPLICATION.Simulation[nProcess].StationFirst  := 2;
      GVL_APPLICATION.Simulation[nProcess].StationLast   := 2;

      GVL_APPLICATION.Simulation[nProcess].TargetFirst   := 3;
      GVL_APPLICATION.Simulation[nProcess].TargetLast    := 3;
      GVL_APPLICATION.Simulation[nProcess].TargetMask    := 2#0011; // mask for target station

      GVL_APPLICATION.Simulation[nProcess].CheckRangeLow := 100.0;
      GVL_APPLICATION.Simulation[nProcess].CheckRangeHigh:= 600.0;

      //---------------------------------------------------------
      nProcess                                        := 2;
      tProcess[nProcess]                              := T#250MS;

      GVL_APPLICATION.Simulation[nProcess].StationFirst  := 3;
      GVL_APPLICATION.Simulation[nProcess].StationLast   := 3;

      GVL_APPLICATION.Simulation[nProcess].TargetFirst   := 4;
      GVL_APPLICATION.Simulation[nProcess].TargetLast    := 5;
      GVL_APPLICATION.Simulation[nProcess].TargetMask    := 2#0001; // mask for target station

      GVL_APPLICATION.Simulation[nProcess].CheckRangeLow := 700.0;
      GVL_APPLICATION.Simulation[nProcess].CheckRangeHigh:= 2100.0;

      //---------------------------------------------------------
      nProcess                                        := 3;
      tProcess[nProcess]                              := T#550MS;

      GVL_APPLICATION.Simulation[nProcess].StationFirst  := 4;
      GVL_APPLICATION.Simulation[nProcess].StationLast   := 5;

      GVL_APPLICATION.Simulation[nProcess].TargetFirst   := 6;
      GVL_APPLICATION.Simulation[nProcess].TargetLast    := 7;
      GVL_APPLICATION.Simulation[nProcess].TargetMask    := 2#0001; // mask for target station

      GVL_APPLICATION.Simulation[nProcess].CheckRangeLow := 4000.0;
      GVL_APPLICATION.Simulation[nProcess].CheckRangeHigh:= 5100.0;

      //---------------------------------------------------------
      nProcess                                        := 4;
      tProcess[nProcess]                              := T#500MS;

      GVL_APPLICATION.Simulation[nProcess].StationFirst  := 6;
      GVL_APPLICATION.Simulation[nProcess].StationLast   := 7;

      GVL_APPLICATION.Simulation[nProcess].TargetFirst   := 8;
      GVL_APPLICATION.Simulation[nProcess].TargetLast    := 8;
      GVL_APPLICATION.Simulation[nProcess].TargetMask    := 2#0001; // mask for target station

      GVL_APPLICATION.Simulation[nProcess].CheckRangeLow := 5000.0;
      GVL_APPLICATION.Simulation[nProcess].CheckRangeHigh:= 6100.0;

      //---------------------------------------------------------
      nProcess                                        := 5;
      tProcess[nProcess]                              := T#500MS;

      GVL_APPLICATION.Simulation[nProcess].StationFirst  := 8;
      GVL_APPLICATION.Simulation[nProcess].StationLast   := 8;

      GVL_APPLICATION.Simulation[nProcess].TargetFirst   := 9;
      GVL_APPLICATION.Simulation[nProcess].TargetLast    := 9;
      GVL_APPLICATION.Simulation[nProcess].TargetMask    := 2#0001; // mask for target station

      GVL_APPLICATION.Simulation[nProcess].CheckRangeLow := 8000.0;
      GVL_APPLICATION.Simulation[nProcess].CheckRangeHigh:= 9100.0;

      //---------------------------------------------------------
      nProcess                                        := 6;
      tProcess[nProcess]                              := T#0MS;

      GVL_APPLICATION.Simulation[nProcess].StationFirst  := 9;
      GVL_APPLICATION.Simulation[nProcess].StationLast   := 9;

      GVL_APPLICATION.Simulation[nProcess].TargetFirst   := 10;
      GVL_APPLICATION.Simulation[nProcess].TargetLast    := 11;
      GVL_APPLICATION.Simulation[nProcess].TargetMask    := 2#0001; // mask for target station

      GVL_APPLICATION.Simulation[nProcess].CheckRangeLow := 9900.0;
      GVL_APPLICATION.Simulation[nProcess].CheckRangeHigh:= 10100.0;

      //---------------------------------------------------------
      nProcess                                        := 7;
      tProcess[nProcess]                              := T#600MS;

      GVL_APPLICATION.Simulation[nProcess].StationFirst  := 10;
      GVL_APPLICATION.Simulation[nProcess].StationLast   := 11;

      GVL_APPLICATION.Simulation[nProcess].TargetFirst   := 12;
      GVL_APPLICATION.Simulation[nProcess].TargetLast    := 13;
      GVL_APPLICATION.Simulation[nProcess].TargetMask    := 2#0001; // mask for target station

      GVL_APPLICATION.Simulation[nProcess].CheckRangeLow := 10900.0;
      GVL_APPLICATION.Simulation[nProcess].CheckRangeHigh:= 11100.0;

      //---------------------------------------------------------
      nProcess                                        := 8;
      tProcess[nProcess]                              := T#550MS;

      GVL_APPLICATION.Simulation[nProcess].StationFirst  := 12;
      GVL_APPLICATION.Simulation[nProcess].StationLast   := 13;

      GVL_APPLICATION.Simulation[nProcess].TargetFirst   := 14;
      GVL_APPLICATION.Simulation[nProcess].TargetLast    := 15;
      GVL_APPLICATION.Simulation[nProcess].TargetMask    := 2#0001; // mask for target station

      GVL_APPLICATION.Simulation[nProcess].CheckRangeLow := 11900.0;
      GVL_APPLICATION.Simulation[nProcess].CheckRangeHigh:= 12100.0;

      //---------------------------------------------------------
      nProcess                                        := 9;
      tProcess[nProcess]                              := T#600MS;

      GVL_APPLICATION.Simulation[nProcess].StationFirst  := 14;
      GVL_APPLICATION.Simulation[nProcess].StationLast   := 15;

      GVL_APPLICATION.Simulation[nProcess].TargetFirst   := 16;
      GVL_APPLICATION.Simulation[nProcess].TargetLast    := 17;
      GVL_APPLICATION.Simulation[nProcess].TargetMask    := 2#0001; // mask for target station

      GVL_APPLICATION.Simulation[nProcess].CheckRangeLow := 13900.0;
      GVL_APPLICATION.Simulation[nProcess].CheckRangeHigh:= 14100.0;

      //---------------------------------------------------------
      nProcess                                        := 10;
      tProcess[nProcess]                              := T#500MS;

      GVL_APPLICATION.Simulation[nProcess].StationFirst  := 16;
      GVL_APPLICATION.Simulation[nProcess].StationLast   := 17;

      GVL_APPLICATION.Simulation[nProcess].TargetFirst   := 18;
      GVL_APPLICATION.Simulation[nProcess].TargetLast    := 19;
      GVL_APPLICATION.Simulation[nProcess].TargetMask    := 2#0001; // mask for target station

      GVL_APPLICATION.Simulation[nProcess].CheckRangeLow := 16900.0;
      GVL_APPLICATION.Simulation[nProcess].CheckRangeHigh:= 17100.0;

      //---------------------------------------------------------
      nProcess                                        := 11;
      tProcess[nProcess]                              := T#100MS;

      GVL_APPLICATION.Simulation[nProcess].StationFirst  := 18;
      GVL_APPLICATION.Simulation[nProcess].StationLast   := 19;

      GVL_APPLICATION.Simulation[nProcess].TargetFirst   := 20;
      GVL_APPLICATION.Simulation[nProcess].TargetLast    := 21;
      GVL_APPLICATION.Simulation[nProcess].TargetMask    := 2#0001; // mask for target station

      GVL_APPLICATION.Simulation[nProcess].CheckRangeLow := 17900.0;
      GVL_APPLICATION.Simulation[nProcess].CheckRangeHigh:= 18100.0;

      //---------------------------------------------------------
      nProcess                                        := 12;
      tProcess[nProcess]                              := T#200MS;

      GVL_APPLICATION.Simulation[nProcess].StationFirst  := 20;
      GVL_APPLICATION.Simulation[nProcess].StationLast   := 21;

      GVL_APPLICATION.Simulation[nProcess].TargetFirst   := 1;
      GVL_APPLICATION.Simulation[nProcess].TargetLast    := 1;
      GVL_APPLICATION.Simulation[nProcess].TargetMask    := 2#0001; // mask for target station

      GVL_APPLICATION.Simulation[nProcess].CheckRangeLow := 19900.0;
      GVL_APPLICATION.Simulation[nProcess].CheckRangeHigh:= 20100.0;

      //---------------------------------------------------------
      nProcess                                        := 13;
      tProcess[nProcess]                              := T#0MS;

      GVL_APPLICATION.Simulation[nProcess].StationFirst  := 1;
      GVL_APPLICATION.Simulation[nProcess].StationLast   := 1;

      GVL_APPLICATION.Simulation[nProcess].TargetFirst   := 2;
      GVL_APPLICATION.Simulation[nProcess].TargetLast    := 2;
      GVL_APPLICATION.Simulation[nProcess].TargetMask    := 2#0001; // mask for target station

      GVL_APPLICATION.Simulation[nProcess].CheckRangeLow := 20900.0;
      GVL_APPLICATION.Simulation[nProcess].CheckRangeHigh:= 21100.0;

    eInit                               := E_PROGRESS.PROGRESS_DONE;

END_CASE
END_ACTION

END_PROGRAM

// ---- _types/f_GetState.TcPOU
// global function to extract state identifier from combined value
FUNCTION f_GetState : uint
VAR_INPUT
  state     : UINT; // combined value of identifier + e_progress
END_VAR
VAR
  _stx      : uint;
END_VAR

_stx          := state MOD E_PROGRESS.PROGRESS_INIT;

IF (_stx = 0)
THEN
  f_GetState  := state;
ELSE
  f_GetState  := _stx;
END_IF

END_FUNCTION

// ---- _types/f_GetProgress.TcPOU
// global function to extract e_progress from combined value
FUNCTION f_GetProgress : uint
VAR_INPUT
  state     : UINT;
END_VAR
VAR
  nP        : uint;
END_VAR


nP := state / E_PROGRESS.PROGRESS_INIT;

f_GetProgress := nP * E_PROGRESS.PROGRESS_INIT;

END_FUNCTION

// ---- _XML/Configuration/fb_Configuration.TcPOU
//---------------------------------------------------------------------------------------------------------------
//
//  fb_Configuration
//
//  HAUD 2023.04.14
//  - base xml integration
//
//  HAUD 2026.04.10.
//  - now extending a base class
//
//  - cyclic OnChange wrapper for xml data 
//      - Ctrl/State
//        1. INIT
//        2. READ / WRITE
//
//  - read  ST_STATION_PARAMETER on demand
//  - write ST_STATION_PARAMETER on demand
//
//---------------------------------------------------------------------------------------------------------------
// This SOFTWARE is provided as an Example by THE PROVIDER "as is" and "with all faults." THE PROVIDER makes no 
// representations or warranties of any kind concerning the safety, suitability, lack of viruses, inaccuracies, 
// typographical errors, or other harmful components of this SOFTWARE. There are inherent dangers in the use of 
// any software, and you are solely responsible for determining whether this SOFTWARE is compatible with your 
// equipment and other software installed on your equipment. You are also solely responsible for the protection 
// of your equipment and backup of your data, and THE PROVIDER will not be liable for any damages you may suffer 
// in connection with using, modifying, or distributing this SOFTWARE.
//---------------------------------------------------------------------------------------------------------------
FUNCTION_BLOCK fb_Configuration EXTENDS fb_XmlBase
VAR
  _stCtrl               : REFERENCE TO ST_DATA_CTRL;
  _stState              : REFERENCE TO ST_DATA_STATE;

  _stConfiguration      : ST_Configuration;
  _pStationParameter    : POINTER TO ARRAY[1..MAX_STATION] OF ST_STATION_PARAMETER;
END_VAR
VAR CONSTANT
  FILE_ROOT             : STRING := 'CONFIG_XtsTransport_';
  X_PATH                : STRING := '/XtsTransport/config';
END_VAR

//---------------------------------------------------------------------------------------------------------------
//  check pointers from the outside
//---------------------------------------------------------------------------------------------------------------
IF NOT Check() THEN RETURN; END_IF
//---------------------------------------------------------------------------------------------------------------
// always build the internal data pointer
//  - as always: better safe than sorry
//  - leave this bit here, it doesn't cost much and safely addresses the data
//---------------------------------------------------------------------------------------------------------------
_pData                        := ADR    (_stConfiguration);
_nData                        := SIZEOF (_stConfiguration);
_sXpath                       := X_PATH;

// copy to local for debug
_eCmd                         := _stCtrl.Cmd;

// cyclic check for command change
// get state for cmd
IF (_eCmd <> _eCmdOld)
THEN
  // get matching sdtate for Ctrl.Cmd
  _eState                     := Cmd(_eCmd);
  _eCmdOld                    := _eCmd;
END_IF


CASE _eResult
OF
  E_PROGRESS.PROGRESS_INVALID:
    _stState.State            := E_DATA_STATE.NULL;

  E_PROGRESS.PROGRESS_ERROR:
    _stState.State            := _eState + E_PROGRESS.PROGRESS_ERROR;

  E_PROGRESS.PROGRESS_DONE:
    _stState.State            := _eState + E_PROGRESS.PROGRESS_DONE;

ELSE
  // work in progress
  // update progress for extern use
  _stState.State              := _eState + _eResult;

  CASE _eState
  OF
    E_DATA_STATE.INIT:
      _eResult   := _eInit    := CreateFolder(TRUE);

    E_DATA_STATE.READ:
      _eResult                := XmlRead(TRUE);
      IF (_eResult = E_PROGRESS.PROGRESS_DONE)
      THEN
        // copy the single ladies
        memcpy(_pStationParameter, ADR(_stConfiguration.XtsStationParameter), SIZEOF(_stConfiguration.XtsStationParameter));
      END_IF

    E_DATA_STATE.WRITE:
      _eResult                := XmlWrite(TRUE);
  ELSE
      _eResult                := E_PROGRESS.PROGRESS_INVALID;
  END_CASE
END_CASE

METHOD Check : BOOL
//-------------------------------------------------------------------------
IF NOT (__ISVALIDREF(_stCtrl))
THEN
  _eCheck               := E_DATA_CHECK.REFERENCE_CTRL_INVALID;
  RETURN;
END_IF
//-------------------------------------------------------------------------
IF NOT (__ISVALIDREF(_stState))
THEN
  _eCheck               := E_DATA_CHECK.REFERENCE_STATE_INVALID;
  RETURN;
END_IF
//-------------------------------------------------------------------------
IF NOT (_pStationParameter <> 0)
THEN
  _eCheck               := E_DATA_CHECK.POINTER_STATION_PARAMETER_INVALID;
  RETURN;
END_IF
//-------------------------------------------------------------------------
_eCheck                 := E_DATA_CHECK.DONE_CHECK;
Check                   := TRUE;
END_METHOD

METHOD PRIVATE Cmd : E_DATA_STATE
VAR_INPUT
  Ctrl      : E_DATA_CTRL;
END_VAR
VAR_INST
  _eState   : E_DATA_STATE;
END_VAR
IF NOT Check() THEN Cmd   := E_DATA_STATE.NULL;  RETURN; END_IF

CASE Ctrl
OF
  //---------------------------------------------------------------
  E_DATA_CTRL.INIT:
    _sName                := concat(FILE_ROOT, _sIdentity);
    _sName                := concat(_sName, '.xml');
    _sFilePath            := concat(_sDirectoryPath, _sName);

